LIN {X 0.103,Y -553.727,Z 590.333,A 0.000,B 0.000,C 90.000,E1 275.853} C_DIS
LIN {X 0.163,Y -552.917,Z 590.320,A 0.000,B 0.000,C 90.000,E1 273.612} C_DIS
LIN {X 0.102,Y -552.398,Z 590.309,A 0.000,B 0.000,C 90.000,E1 271.661} C_DIS
LIN {X -0.195,Y -552.147,Z 590.303,A 0.000,B 0.000,C 90.000,E1 270.573} C_DIS
LIN {X 0.184,Y -551.566,Z 590.294,A 0.000,B 0.000,C 90.000,E1 268.854} C_DIS
LIN {X 0.006,Y -550.867,Z 590.284,A 0.000,B 0.000,C 90.000,E1 267.192} C_DIS
LIN {X -0.206,Y -550.289,Z 590.277,A 0.000,B 0.000,C 90.000,E1 265.812} C_DIS
LIN {X 0.126,Y -549.551,Z 590.269,A 0.000,B 0.000,C 90.000,E1 264.375} C_DIS
LIN {X -0.148,Y -548.851,Z 590.263,A 0.000,B 0.000,C 90.000,E1 263.280} C_DIS
LIN {X 0.107,Y -547.994,Z 590.256,A 0.000,B 0.000,C 90.000,E1 262.129} C_DIS
LIN {X -0.025,Y -546.676,Z 590.249,A 0.000,B 0.000,C 90.000,E1 260.735} C_DIS
LIN {X 0.008,Y -544.774,Z 590.238,A 0.000,B 0.000,C 90.000,E1 258.757} C_DIS
LIN {X -0.079,Y -543.391,Z 590.230,A 0.000,B 0.000,C 90.000,E1 257.353} C_DIS
LIN {X 0.294,Y -541.048,Z 590.217,A 0.000,B 0.000,C 90.000,E1 255.046} C_DIS
LIN {X -0.049,Y -539.330,Z 590.208,A 0.000,B 0.000,C 90.000,E1 253.378} C_DIS
LIN {X 0.028,Y -537.748,Z 590.200,A 0.000,B 0.000,C 90.000,E1 251.945} C_DIS
LIN {X 0.200,Y -536.335,Z 590.193,A 0.000,B 0.000,C 90.000,E1 250.786} C_DIS
LIN {X 0.172,Y -534.674,Z 590.187,A 0.000,B 0.000,C 90.000,E1 249.645} C_DIS
LIN {X 0.288,Y -533.258,Z 590.182,A 0.000,B 0.000,C 90.000,E1 248.773} C_DIS
LIN {X 0.092,Y -530.601,Z 590.174,A 0.000,B 0.000,C 90.000,E1 247.358} C_DIS
LIN {X 0.227,Y -527.112,Z 590.165,A 0.000,B 0.000,C 90.000,E1 245.613} C_DIS
LIN {X 0.176,Y -524.691,Z 590.158,A 0.000,B 0.000,C 90.000,E1 244.460} C_DIS
LIN {X 0.245,Y -521.535,Z 590.150,A 0.000,B 0.000,C 90.000,E1 242.999} C_DIS
LIN {X 0.030,Y -518.163,Z 590.142,A 0.000,B 0.000,C 90.000,E1 241.563} C_DIS
LIN {X 0.098,Y -515.229,Z 590.136,A 0.000,B 0.000,C 90.000,E1 240.383} C_DIS
LIN {X 0.011,Y -509.881,Z 590.124,A 0.000,B 0.000,C 90.000,E1 238.329} C_DIS
LIN {X 0.105,Y -506.106,Z 590.116,A 0.000,B 0.000,C 90.000,E1 236.834} C_DIS
LIN {X -0.183,Y -502.744,Z 590.109,A 0.000,B 0.000,C 90.000,E1 235.674} C_DIS
LIN {X -0.116,Y -500.117,Z 590.104,A 0.000,B 0.000,C 90.000,E1 234.769} C_DIS
LIN {X 0.097,Y -492.736,Z 590.089,A 0.000,B 0.000,C 90.000,E1 232.029} C_DIS
LIN {X 0.027,Y -488.658,Z 590.081,A 0.000,B 0.000,C 90.000,E1 230.517} C_DIS
LIN {X -0.190,Y -484.697,Z 590.072,A 0.000,B 0.000,C 90.000,E1 229.013} C_DIS
LIN {X 0.093,Y -479.290,Z 590.060,A 0.000,B 0.000,C 90.000,E1 226.824} C_DIS
LIN {X -0.217,Y -474.782,Z 590.050,A 0.000,B 0.000,C 90.000,E1 225.000} C_DIS
LIN {X 0.185,Y -471.918,Z 590.043,A 0.000,B 0.000,C 90.000,E1 223.704} C_DIS
LIN {X 0.050,Y -467.520,Z 590.033,A 0.000,B 0.000,C 90.000,E1 221.838} C_DIS
LIN {X 0.112,Y -464.046,Z 590.024,A 0.000,B 0.000,C 90.000,E1 220.253} C_DIS
LIN {X 0.102,Y -460.700,Z 590.015,A 0.000,B 0.000,C 90.000,E1 218.669} C_DIS
LIN {X 0.094,Y -457.363,Z 590.006,A 0.000,B 0.000,C 90.000,E1 217.076} C_DIS
LIN {X -0.154,Y -453.442,Z 589.995,A 0.000,B 0.000,C 90.000,E1 215.185} C_DIS
LIN {X -0.110,Y -449.724,Z 589.985,A 0.000,B 0.000,C 90.000,E1 213.245} C_DIS
LIN {X -0.138,Y -443.891,Z 589.967,A 0.000,B 0.000,C 90.000,E1 210.001} C_DIS
LIN {X -0.203,Y -439.747,Z 589.954,A 0.000,B 0.000,C 90.000,E1 207.719} C_DIS
LIN {X -0.042,Y -436.870,Z 589.945,A 0.000,B 0.000,C 90.000,E1 206.052} C_DIS
LIN {X 0.098,Y -432.893,Z 589.932,A 0.000,B 0.000,C 90.000,E1 203.718} C_DIS
LIN {X 0.158,Y -428.613,Z 589.917,A 0.000,B 0.000,C 90.000,E1 201.046} C_DIS
LIN {X 0.166,Y -424.518,Z 589.902,A 0.000,B 0.000,C 90.000,E1 198.362} C_DIS
LIN {X 0.174,Y -420.785,Z 589.887,A 0.000,B 0.000,C 90.000,E1 195.662} C_DIS
LIN {X -0.186,Y -419.030,Z 589.880,A 0.000,B 0.000,C 90.000,E1 194.356} C_DIS
LIN {X 0.141,Y -417.098,Z 589.872,A 0.000,B 0.000,C 90.000,E1 192.952} C_DIS
LIN {X -0.146,Y -413.611,Z 589.859,A 0.000,B 0.000,C 90.000,E1 190.602} C_DIS
LIN {X 0.151,Y -410.179,Z 589.844,A 0.000,B 0.000,C 90.000,E1 187.814} C_DIS
LIN {X 0.197,Y -408.564,Z 589.836,A 0.000,B 0.000,C 90.000,E1 186.429} C_DIS
LIN {X 0.098,Y -404.784,Z 589.819,A 0.000,B 0.000,C 90.000,E1 183.326} C_DIS
LIN {X 0.160,Y -401.368,Z 589.797,A 0.000,B 0.000,C 90.000,E1 179.484} C_DIS
LIN {X -0.165,Y -399.570,Z 589.782,A 0.000,B 0.000,C 90.000,E1 176.731} C_DIS
LIN {X -0.089,Y -398.435,Z 589.766,A 0.000,B 0.000,C 90.000,E1 173.913} C_DIS
LIN {X 0.009,Y -397.785,Z 589.749,A 0.000,B 0.000,C 90.000,E1 170.735} C_DIS
LIN {X -0.126,Y -397.766,Z 589.731,A 0.000,B 0.000,C 90.000,E1 167.589} C_DIS
LIN {X 0.052,Y -398.187,Z 589.717,A 0.000,B 0.000,C 90.000,E1 165.102} C_DIS
LIN {X -0.064,Y -398.968,Z 589.702,A 0.000,B 0.000,C 90.000,E1 162.308} C_DIS
LIN {X 0.034,Y -399.714,Z 589.690,A 0.000,B 0.000,C 90.000,E1 160.188} C_DIS
LIN {X -0.168,Y -400.409,Z 589.680,A 0.000,B 0.000,C 90.000,E1 158.465} C_DIS
LIN {X -0.120,Y -401.392,Z 589.669,A 0.000,B 0.000,C 90.000,E1 156.357} C_DIS
LIN {X 0.102,Y -402.364,Z 589.657,A 0.000,B 0.000,C 90.000,E1 154.229} C_DIS
LIN {X -0.024,Y -403.383,Z 589.645,A 0.000,B 0.000,C 90.000,E1 152.153} C_DIS
LIN {X -0.024,Y -404.131,Z 589.636,A 0.000,B 0.000,C 90.000,E1 150.411} C_DIS
LIN {X 0.135,Y -404.680,Z 589.628,A 0.000,B 0.000,C 90.000,E1 148.997} C_DIS
LIN {X 0.213,Y -405.235,Z 589.618,A 0.000,B 0.000,C 90.000,E1 147.248} C_DIS
LIN {X 0.086,Y -405.715,Z 589.607,A 0.000,B 0.000,C 90.000,E1 145.182} C_DIS
LIN {X -0.031,Y -406.113,Z 589.597,A 0.000,B 0.000,C 90.000,E1 143.463} C_DIS
LIN {X 0.009,Y -406.580,Z 589.585,A 0.000,B 0.000,C 90.000,E1 141.376} C_DIS
LIN {X 0.156,Y -406.984,Z 589.576,A 0.000,B 0.000,C 90.000,E1 139.622} C_DIS
LIN {X 0.114,Y -407.316,Z 589.568,A 0.000,B 0.000,C 90.000,E1 138.243} C_DIS
LIN {X -0.240,Y -407.605,Z 589.557,A 0.000,B 0.000,C 90.000,E1 136.215} C_DIS
LIN {X 0.134,Y -407.816,Z 589.547,A 0.000,B 0.000,C 90.000,E1 134.433} C_DIS
LIN {X 0.071,Y -408.085,Z 589.535,A 0.000,B 0.000,C 90.000,E1 132.366} C_DIS
LIN {X 0.194,Y -408.172,Z 589.526,A 0.000,B 0.000,C 90.000,E1 130.620} C_DIS
LIN {X -0.092,Y -408.216,Z 589.518,A 0.000,B 0.000,C 90.000,E1 129.277} C_DIS
LIN {X 0.167,Y -408.231,Z 589.514,A 0.000,B 0.000,C 90.000,E1 128.463} C_DIS
LIN {X -0.072,Y -414.947,Z 589.501,A 0.000,B 0.000,C 90.000,E1 126.171} C_DIS
LIN {X 0.101,Y -415.909,Z 589.499,A 0.000,B 0.000,C 90.000,E1 125.804} C_DIS
LIN {X -0.016,Y -425.391,Z 589.478,A 0.000,B 0.000,C 90.000,E1 122.084} C_DIS
LIN {X -0.086,Y -428.983,Z 589.471,A 0.000,B 0.000,C 90.000,E1 120.875} C_DIS
LIN {X -0.125,Y -429.060,Z 589.471,A 0.000,B 0.000,C 90.000,E1 120.875} C_DIS
LIN {X 0.076,Y -438.663,Z 589.469,A 0.000,B 0.000,C 90.000,E1 120.413} C_DIS
LIN {X -0.052,Y -453.951,Z 589.465,A 0.000,B 0.000,C 90.000,E1 119.716} C_DIS
LIN {X 0.129,Y -467.535,Z 589.461,A 0.000,B 0.000,C 90.000,E1 119.027} C_DIS
LIN {X 0.032,Y -475.906,Z 589.459,A 0.000,B 0.000,C 90.000,E1 118.615} C_DIS
LIN {X -0.202,Y -485.846,Z 589.456,A 0.000,B 0.000,C 90.000,E1 118.103} C_DIS
LIN {X -0.052,Y -495.708,Z 589.453,A 0.000,B 0.000,C 90.000,E1 117.513} C_DIS
LIN {X -0.071,Y -502.085,Z 589.451,A 0.000,B 0.000,C 90.000,E1 117.129} C_DIS
LIN {X -0.060,Y -512.802,Z 589.447,A 0.000,B 0.000,C 90.000,E1 116.437} C_DIS
LIN {X 0.057,Y -517.558,Z 589.445,A 0.000,B 0.000,C 90.000,E1 116.104} C_DIS
LIN {X -0.067,Y -526.534,Z 589.441,A 0.000,B 0.000,C 90.000,E1 115.463} C_DIS
LIN {X 0.238,Y -533.686,Z 589.439,A 0.000,B 0.000,C 90.000,E1 114.899} C_DIS
LIN {X -0.150,Y -538.090,Z 589.437,A 0.000,B 0.000,C 90.000,E1 114.591} C_DIS
LIN {X 0.027,Y -544.873,Z 589.433,A 0.000,B 0.000,C 90.000,E1 114.003} C_DIS
LIN {X 0.244,Y -548.783,Z 589.432,A 0.000,B 0.000,C 90.000,E1 113.643} C_DIS
LIN {X -0.013,Y -554.752,Z 589.428,A 0.000,B 0.000,C 90.000,E1 113.078} C_DIS
LIN {X 0.050,Y -559.282,Z 589.426,A 0.000,B 0.000,C 90.000,E1 112.589} C_DIS
LIN {X 0.096,Y -564.684,Z 589.422,A 0.000,B 0.000,C 90.000,E1 111.897} C_DIS
LIN {X -0.075,Y -569.428,Z 589.418,A 0.000,B 0.000,C 90.000,E1 111.227} C_DIS
LIN {X -0.206,Y -573.566,Z 589.414,A 0.000,B 0.000,C 90.000,E1 110.556} C_DIS
LIN {X 0.078,Y -578.598,Z 589.409,A 0.000,B 0.000,C 90.000,E1 109.577} C_DIS
LIN {X -0.131,Y -583.212,Z 589.404,A 0.000,B 0.000,C 90.000,E1 108.652} C_DIS
LIN {X 0.147,Y -586.751,Z 589.399,A 0.000,B 0.000,C 90.000,E1 107.819} C_DIS
LIN {X 0.229,Y -588.912,Z 589.396,A 0.000,B 0.000,C 90.000,E1 107.275} C_DIS
LIN {X 0.009,Y -591.975,Z 589.392,A 0.000,B 0.000,C 90.000,E1 106.496} C_DIS
LIN {X 0.087,Y -595.800,Z 589.386,A 0.000,B 0.000,C 90.000,E1 105.426} C_DIS
LIN {X 0.220,Y -599.376,Z 589.380,A 0.000,B 0.000,C 90.000,E1 104.356} C_DIS
LIN {X 0.023,Y -605.560,Z 589.370,A 0.000,B 0.000,C 90.000,E1 102.535} C_DIS
LIN {X -0.031,Y -611.800,Z 589.360,A 0.000,B 0.000,C 90.000,E1 100.715} C_DIS
LIN {X -0.299,Y -614.429,Z 589.355,A 0.000,B 0.000,C 90.000,E1 99.962} C_DIS
LIN {X 0.196,Y -618.587,Z 589.348,A 0.000,B 0.000,C 90.000,E1 98.624} C_DIS
LIN {X 0.057,Y -622.599,Z 589.341,A 0.000,B 0.000,C 90.000,E1 97.352} C_DIS
LIN {X 0.211,Y -625.609,Z 589.335,A 0.000,B 0.000,C 90.000,E1 96.315} C_DIS
LIN {X 0.012,Y -627.702,Z 589.331,A 0.000,B 0.000,C 90.000,E1 95.568} C_DIS
LIN {X 0.236,Y -630.228,Z 589.325,A 0.000,B 0.000,C 90.000,E1 94.531} C_DIS
LIN {X -0.189,Y -632.360,Z 589.320,A 0.000,B 0.000,C 90.000,E1 93.555} C_DIS
LIN {X -0.214,Y -634.585,Z 589.313,A 0.000,B 0.000,C 90.000,E1 92.293} C_DIS
LIN {X 0.303,Y -635.778,Z 589.308,A 0.000,B 0.000,C 90.000,E1 91.489} C_DIS
LIN {X 0.049,Y -636.150,Z 589.307,A 0.000,B 0.000,C 90.000,E1 91.260} C_DIS
LIN {X 0.065,Y -637.392,Z 589.300,A 0.000,B 0.000,C 90.000,E1 90.000} C_DIS
LIN {X -0.041,Y -637.871,Z 589.296,A 0.000,B 0.000,C 90.000,E1 89.255} C_DIS
LIN {X -0.146,Y -638.129,Z 589.292,A 0.000,B 0.000,C 90.000,E1 88.511} C_DIS
LIN {X -0.229,Y -638.123,Z 589.288,A 0.000,B 0.000,C 90.000,E1 87.764} C_DIS
LIN {X 0.300,Y -637.875,Z 589.283,A 0.000,B 0.000,C 90.000,E1 86.963} C_DIS
LIN {X -0.034,Y -637.318,Z 589.278,A 0.000,B 0.000,C 90.000,E1 85.988} C_DIS
LIN {X 0.310,Y -636.408,Z 589.272,A 0.000,B 0.000,C 90.000,E1 84.951} C_DIS
LIN {X 0.017,Y -635.312,Z 589.267,A 0.000,B 0.000,C 90.000,E1 83.970} C_DIS
LIN {X -0.088,Y -634.277,Z 589.262,A 0.000,B 0.000,C 90.000,E1 83.223} C_DIS
LIN {X 0.217,Y -632.525,Z 589.257,A 0.000,B 0.000,C 90.000,E1 82.186} C_DIS
LIN {X -0.041,Y -630.463,Z 589.251,A 0.000,B 0.000,C 90.000,E1 81.197} C_DIS
LIN {X 0.302,Y -628.200,Z 589.245,A 0.000,B 0.000,C 90.000,E1 80.151} C_DIS
LIN {X -0.006,Y -625.708,Z 589.240,A 0.000,B 0.000,C 90.000,E1 79.162} C_DIS
LIN {X 0.046,Y -622.308,Z 589.233,A 0.000,B 0.000,C 90.000,E1 77.881} C_DIS
LIN {X 0.222,Y -620.910,Z 589.230,A 0.000,B 0.000,C 90.000,E1 77.353} C_DIS
LIN {X -0.286,Y -617.015,Z 589.223,A 0.000,B 0.000,C 90.000,E1 76.117} C_DIS
LIN {X -0.229,Y -614.491,Z 589.219,A 0.000,B 0.000,C 90.000,E1 75.338} C_DIS
LIN {X -0.005,Y -610.833,Z 589.213,A 0.000,B 0.000,C 90.000,E1 74.283} C_DIS
LIN {X -0.264,Y -606.705,Z 589.207,A 0.000,B 0.000,C 90.000,E1 73.268} C_DIS
LIN {X -0.304,Y -603.342,Z 589.203,A 0.000,B 0.000,C 90.000,E1 72.489} C_DIS
LIN {X -0.145,Y -600.317,Z 589.199,A 0.000,B 0.000,C 90.000,E1 71.819} C_DIS
LIN {X 0.202,Y -594.996,Z 589.193,A 0.000,B 0.000,C 90.000,E1 70.732} C_DIS
LIN {X 0.228,Y -590.658,Z 589.189,A 0.000,B 0.000,C 90.000,E1 69.934} C_DIS
LIN {X 0.013,Y -585.840,Z 589.184,A 0.000,B 0.000,C 90.000,E1 69.156} C_DIS
LIN {X 0.227,Y -581.416,Z 589.181,A 0.000,B 0.000,C 90.000,E1 68.465} C_DIS
LIN {X -0.271,Y -577.630,Z 589.178,A 0.000,B 0.000,C 90.000,E1 67.975} C_DIS
LIN {X -0.025,Y -572.375,Z 589.174,A 0.000,B 0.000,C 90.000,E1 67.283} C_DIS
LIN {X -0.251,Y -566.931,Z 589.170,A 0.000,B 0.000,C 90.000,E1 66.666} C_DIS
LIN {X 0.142,Y -563.380,Z 589.168,A 0.000,B 0.000,C 90.000,E1 66.230} C_DIS
LIN {X 0.231,Y -557.214,Z 589.165,A 0.000,B 0.000,C 90.000,E1 65.613} C_DIS
LIN {X -0.039,Y -552.060,Z 589.162,A 0.000,B 0.000,C 90.000,E1 65.177} C_DIS
LIN {X 0.031,Y -546.519,Z 589.160,A 0.000,B 0.000,C 90.000,E1 64.717} C_DIS
LIN {X -0.316,Y -541.738,Z 589.158,A 0.000,B 0.000,C 90.000,E1 64.409} C_DIS
LIN {X -0.139,Y -536.929,Z 589.156,A 0.000,B 0.000,C 90.000,E1 64.076} C_DIS
LIN {X 0.261,Y -530.053,Z 589.154,A 0.000,B 0.000,C 90.000,E1 63.640} C_DIS
LIN {X 0.086,Y -523.161,Z 589.152,A 0.000,B 0.000,C 90.000,E1 63.307} C_DIS
LIN {X -0.078,Y -516.360,Z 589.150,A 0.000,B 0.000,C 90.000,E1 62.999} C_DIS
LIN {X -0.092,Y -505.953,Z 589.147,A 0.000,B 0.000,C 90.000,E1 62.538} C_DIS
LIN {X -0.103,Y -492.338,Z 589.144,A 0.000,B 0.000,C 90.000,E1 61.948} C_DIS
LIN {X -0.006,Y -458.334,Z 589.136,A 0.000,B 0.000,C 90.000,E1 60.411} C_DIS
LIN {X -0.122,Y -450.998,Z 589.134,A 0.000,B 0.000,C 90.000,E1 60.049} C_DIS
LIN {X 0.226,Y -450.975,Z 589.134,A 0.000,B 0.000,C 90.000,E1 59.999} C_DIS
LIN {X 0.224,Y -444.233,Z 589.115,A 0.000,B 0.000,C 90.000,E1 56.628} C_DIS
LIN {X -0.087,Y -443.543,Z 589.113,A 0.000,B 0.000,C 90.000,E1 56.342} C_DIS
LIN {X -0.075,Y -434.458,Z 589.091,A 0.000,B 0.000,C 90.000,E1 52.396} C_DIS
LIN {X -0.070,Y -433.807,Z 589.089,A 0.000,B 0.000,C 90.000,E1 52.065} C_DIS
LIN {X -0.108,Y -433.823,Z 589.088,A 0.000,B 0.000,C 90.000,E1 51.904} C_DIS
LIN {X -0.028,Y -435.444,Z 589.078,A 0.000,B 0.000,C 90.000,E1 50.070} C_DIS
LIN {X 0.005,Y -437.214,Z 589.067,A 0.000,B 0.000,C 90.000,E1 48.081} C_DIS
LIN {X -0.011,Y -439.520,Z 589.052,A 0.000,B 0.000,C 90.000,E1 45.445} C_DIS
LIN {X 0.155,Y -440.657,Z 589.045,A 0.000,B 0.000,C 90.000,E1 44.109} C_DIS
LIN {X 0.022,Y -441.542,Z 589.038,A 0.000,B 0.000,C 90.000,E1 42.813} C_DIS
LIN {X -0.077,Y -442.261,Z 589.031,A 0.000,B 0.000,C 90.000,E1 41.515} C_DIS
LIN {X -0.130,Y -442.741,Z 589.025,A 0.000,B 0.000,C 90.000,E1 40.539} C_DIS
LIN {X -0.186,Y -443.365,Z 589.016,A 0.000,B 0.000,C 90.000,E1 38.910} C_DIS
LIN {X 0.119,Y -443.853,Z 589.007,A 0.000,B 0.000,C 90.000,E1 37.237} C_DIS
LIN {X -0.193,Y -444.089,Z 589.002,A 0.000,B 0.000,C 90.000,E1 36.297} C_DIS
LIN {X 0.214,Y -444.268,Z 588.992,A 0.000,B 0.000,C 90.000,E1 34.612} C_DIS
LIN {X 0.000,Y -444.218,Z 588.983,A 0.000,B 0.000,C 90.000,E1 33.007} C_DIS
LIN {X 0.027,Y -444.239,Z 588.971,A 0.000,B 0.000,C 90.000,E1 30.718} C_DIS
LIN {X 0.097,Y -444.213,Z 588.962,A 0.000,B 0.000,C 90.000,E1 29.077} C_DIS
LIN {X 0.012,Y -444.260,Z 588.951,A 0.000,B 0.000,C 90.000,E1 27.129} C_DIS
LIN {X -0.179,Y -444.308,Z 588.944,A 0.000,B 0.000,C 90.000,E1 25.848} C_DIS
LIN {X -0.112,Y -444.484,Z 588.934,A 0.000,B 0.000,C 90.000,E1 24.207} C_DIS
LIN {X -0.219,Y -444.728,Z 588.925,A 0.000,B 0.000,C 90.000,E1 22.589} C_DIS
LIN {X -0.047,Y -445.056,Z 588.914,A 0.000,B 0.000,C 90.000,E1 20.610} C_DIS
LIN {X 0.104,Y -445.449,Z 588.902,A 0.000,B 0.000,C 90.000,E1 18.308} C_DIS
LIN {X 0.132,Y -446.068,Z 588.889,A 0.000,B 0.000,C 90.000,E1 16.024} C_DIS
LIN {X -0.072,Y -446.918,Z 588.877,A 0.000,B 0.000,C 90.000,E1 13.772} C_DIS
LIN {X -0.180,Y -448.284,Z 588.862,A 0.000,B 0.000,C 90.000,E1 11.186} C_DIS
LIN {X 0.016,Y -449.845,Z 588.848,A 0.000,B 0.000,C 90.000,E1 8.568} C_DIS
LIN {X 0.122,Y -451.773,Z 588.833,A 0.000,B 0.000,C 90.000,E1 5.967} C_DIS
LIN {X 0.160,Y -454.081,Z 588.819,A 0.000,B 0.000,C 90.000,E1 3.383} C_DIS
LIN {X 0.070,Y -456.397,Z 588.806,A 0.000,B 0.000,C 90.000,E1 1.146} C_DIS
LIN {X -0.166,Y -459.209,Z 588.794,A 0.000,B 0.000,C 90.000,E1 358.854} C_DIS
LIN {X 0.091,Y -462.759,Z 588.779,A 0.000,B 0.000,C 90.000,E1 356.274} C_DIS
LIN {X -0.193,Y -466.009,Z 588.767,A 0.000,B 0.000,C 90.000,E1 354.090} C_DIS
LIN {X -0.104,Y -468.966,Z 588.757,A 0.000,B 0.000,C 90.000,E1 352.186} C_DIS
LIN {X 0.117,Y -471.829,Z 588.746,A 0.000,B 0.000,C 90.000,E1 350.274} C_DIS
LIN {X 0.019,Y -474.779,Z 588.736,A 0.000,B 0.000,C 90.000,E1 348.409} C_DIS
LIN {X 0.082,Y -477.877,Z 588.725,A 0.000,B 0.000,C 90.000,E1 346.533} C_DIS
LIN {X 0.011,Y -480.559,Z 588.717,A 0.000,B 0.000,C 90.000,E1 344.991} C_DIS
LIN {X -0.016,Y -484.658,Z 588.705,A 0.000,B 0.000,C 90.000,E1 342.834} C_DIS
LIN {X 0.082,Y -489.289,Z 588.691,A 0.000,B 0.000,C 90.000,E1 340.369} C_DIS
LIN {X 0.057,Y -492.236,Z 588.683,A 0.000,B 0.000,C 90.000,E1 338.847} C_DIS
LIN {X -0.148,Y -495.533,Z 588.672,A 0.000,B 0.000,C 90.000,E1 337.050} C_DIS
LIN {X -0.139,Y -498.127,Z 588.664,A 0.000,B 0.000,C 90.000,E1 335.537} C_DIS
LIN {X -0.141,Y -500.051,Z 588.657,A 0.000,B 0.000,C 90.000,E1 334.332} C_DIS
LIN {X -0.117,Y -501.996,Z 588.651,A 0.000,B 0.000,C 90.000,E1 333.127} C_DIS
LIN {X 0.025,Y -505.703,Z 588.637,A 0.000,B 0.000,C 90.000,E1 330.717} C_DIS
LIN {X -0.243,Y -508.962,Z 588.626,A 0.000,B 0.000,C 90.000,E1 328.663} C_DIS
LIN {X 0.196,Y -511.902,Z 588.616,A 0.000,B 0.000,C 90.000,E1 326.834} C_DIS
LIN {X 0.195,Y -515.529,Z 588.604,A 0.000,B 0.000,C 90.000,E1 324.769} C_DIS
LIN {X 0.154,Y -519.390,Z 588.593,A 0.000,B 0.000,C 90.000,E1 322.718} C_DIS
LIN {X -0.344,Y -523.881,Z 588.580,A 0.000,B 0.000,C 90.000,E1 320.436} C_DIS
LIN {X 0.128,Y -526.920,Z 588.572,A 0.000,B 0.000,C 90.000,E1 318.933} C_DIS
LIN {X -0.027,Y -529.247,Z 588.567,A 0.000,B 0.000,C 90.000,E1 318.081} C_DIS
LIN {X -0.322,Y -531.709,Z 588.563,A 0.000,B 0.000,C 90.000,E1 317.391} C_DIS
LIN {X -0.116,Y -534.196,Z 588.561,A 0.000,B 0.000,C 90.000,E1 316.905} C_DIS
LIN {X 0.070,Y -536.378,Z 588.559,A 0.000,B 0.000,C 90.000,E1 316.581} C_DIS
LIN {X 0.054,Y -538.214,Z 588.557,A 0.000,B 0.000,C 90.000,E1 316.296} C_DIS
LIN {X -0.273,Y -542.054,Z 588.555,A 0.000,B 0.000,C 90.000,E1 315.891} C_DIS
LIN {X 0.136,Y -546.676,Z 588.552,A 0.000,B 0.000,C 90.000,E1 315.405} C_DIS
LIN {X -0.087,Y -551.915,Z 588.550,A 0.000,B 0.000,C 90.000,E1 315.000} C_DIS
LIN {X 0.208,Y -566.862,Z 588.544,A 0.000,B 0.000,C 90.000,E1 313.866} C_DIS
LIN {X 0.158,Y -587.500,Z 588.536,A 0.000,B 0.000,C 90.000,E1 312.366} C_DIS
LIN {X -0.077,Y -593.270,Z 588.533,A 0.000,B 0.000,C 90.000,E1 311.962} C_DIS
LIN {X 0.100,Y -600.352,Z 588.530,A 0.000,B 0.000,C 90.000,E1 311.391} C_DIS
LIN {X -0.078,Y -604.427,Z 588.528,A 0.000,B 0.000,C 90.000,E1 311.067} C_DIS
LIN {X 0.064,Y -610.932,Z 588.525,A 0.000,B 0.000,C 90.000,E1 310.458} C_DIS
LIN {X 0.040,Y -613.520,Z 588.523,A 0.000,B 0.000,C 90.000,E1 310.216} C_DIS
LIN {X -0.290,Y -619.311,Z 588.520,A 0.000,B 0.000,C 90.000,E1 309.644} C_DIS
LIN {X 0.137,Y -623.800,Z 588.517,A 0.000,B 0.000,C 90.000,E1 309.116} C_DIS
LIN {X -0.138,Y -630.493,Z 588.513,A 0.000,B 0.000,C 90.000,E1 308.382} C_DIS
LIN {X -0.048,Y -638.673,Z 588.508,A 0.000,B 0.000,C 90.000,E1 307.363} C_DIS
LIN {X -0.155,Y -642.541,Z 588.505,A 0.000,B 0.000,C 90.000,E1 306.870} C_DIS
LIN {X -0.235,Y -646.121,Z 588.502,A 0.000,B 0.000,C 90.000,E1 306.377} C_DIS
LIN {X -0.190,Y -651.020,Z 588.498,A 0.000,B 0.000,C 90.000,E1 305.644} C_DIS
LIN {X 0.318,Y -654.104,Z 588.495,A 0.000,B 0.000,C 90.000,E1 305.105} C_DIS
LIN {X 0.275,Y -656.265,Z 588.493,A 0.000,B 0.000,C 90.000,E1 304.739} C_DIS
LIN {X 0.332,Y -659.571,Z 588.490,A 0.000,B 0.000,C 90.000,E1 304.119} C_DIS
LIN {X -0.003,Y -662.000,Z 588.487,A 0.000,B 0.000,C 90.000,E1 303.658} C_DIS
LIN {X -0.393,Y -665.301,Z 588.483,A 0.000,B 0.000,C 90.000,E1 302.959} C_DIS
LIN {X -0.197,Y -668.414,Z 588.479,A 0.000,B 0.000,C 90.000,E1 302.212} C_DIS
LIN {X 0.189,Y -672.332,Z 588.474,A 0.000,B 0.000,C 90.000,E1 301.209} C_DIS
LIN {X 0.047,Y -676.130,Z 588.468,A 0.000,B 0.000,C 90.000,E1 300.256} C_DIS
LIN {X 0.197,Y -679.703,Z 588.463,A 0.000,B 0.000,C 90.000,E1 299.283} C_DIS
LIN {X -0.199,Y -683.002,Z 588.458,A 0.000,B 0.000,C 90.000,E1 298.359} C_DIS
LIN {X 0.262,Y -686.713,Z 588.451,A 0.000,B 0.000,C 90.000,E1 297.129} C_DIS
LIN {X 0.014,Y -688.584,Z 588.447,A 0.000,B 0.000,C 90.000,E1 296.437} C_DIS
LIN {X -0.373,Y -688.952,Z 588.446,A 0.000,B 0.000,C 90.000,E1 296.232} C_DIS
LIN {X 0.089,Y -689.180,Z 588.443,A 0.000,B 0.000,C 90.000,E1 295.720} C_DIS
LIN {X 0.321,Y -688.932,Z 588.442,A 0.000,B 0.000,C 90.000,E1 295.463} C_DIS
LIN {X -0.132,Y -687.243,Z 588.439,A 0.000,B 0.000,C 90.000,E1 295.027} C_DIS
LIN {X -0.018,Y -686.727,Z 588.438,A 0.000,B 0.000,C 90.000,E1 294.899} C_DIS
LIN {X 0.096,Y -685.999,Z 588.438,A 0.000,B 0.000,C 90.000,E1 294.771} C_DIS
LIN {X 0.206,Y -684.865,Z 588.437,A 0.000,B 0.000,C 90.000,E1 294.643} C_DIS
LIN {X 0.313,Y -680.019,Z 588.435,A 0.000,B 0.000,C 90.000,E1 294.207} C_DIS
LIN {X -0.121,Y -678.129,Z 588.434,A 0.000,B 0.000,C 90.000,E1 294.131} C_DIS
LIN {X -0.045,Y -670.038,Z 588.432,A 0.000,B 0.000,C 90.000,E1 293.823} C_DIS
LIN {X -0.184,Y -667.501,Z 588.432,A 0.000,B 0.000,C 90.000,E1 293.770} C_DIS
LIN {X -0.305,Y -661.294,Z 588.431,A 0.000,B 0.000,C 90.000,E1 293.643} C_DIS
LIN {X 0.269,Y -638.978,Z 588.429,A 0.000,B 0.000,C 90.000,E1 293.206} C_DIS
LIN {X -0.018,Y -629.598,Z 588.428,A 0.000,B 0.000,C 90.000,E1 293.025} C_DIS
LIN {X -0.193,Y -616.215,Z 588.426,A 0.000,B 0.000,C 90.000,E1 292.695} C_DIS
LIN {X -0.203,Y -595.903,Z 588.423,A 0.000,B 0.000,C 90.000,E1 292.078} C_DIS
LIN {X 0.143,Y -578.394,Z 588.419,A 0.000,B 0.000,C 90.000,E1 291.482} C_DIS
LIN {X 0.025,Y -571.534,Z 588.418,A 0.000,B 0.000,C 90.000,E1 291.280} C_DIS
LIN {X -0.186,Y -566.448,Z 588.417,A 0.000,B 0.000,C 90.000,E1 291.099} C_DIS
LIN {X 0.220,Y -561.824,Z 588.416,A 0.000,B 0.000,C 90.000,E1 290.791} C_DIS
LIN {X 0.191,Y -561.777,Z 588.416,A 0.000,B 0.000,C 90.000,E1 290.791} C_DIS
LIN {X 0.127,Y -560.661,Z 588.415,A 0.000,B 0.000,C 90.000,E1 290.610} C_DIS
LIN {X 0.085,Y -560.646,Z 588.415,A 0.000,B 0.000,C 90.000,E1 290.610} C_DIS
LIN {X 0.204,Y -560.137,Z 588.412,A 0.000,B 0.000,C 90.000,E1 290.174} C_DIS
LIN {X -0.104,Y -560.141,Z 588.405,A 0.000,B 0.000,C 90.000,E1 288.833} C_DIS
LIN {X 0.222,Y -559.944,Z 588.398,A 0.000,B 0.000,C 90.000,E1 287.692} C_DIS
LIN {X -0.258,Y -559.330,Z 588.389,A 0.000,B 0.000,C 90.000,E1 286.079} C_DIS
LIN {X -0.094,Y -558.821,Z 588.383,A 0.000,B 0.000,C 90.000,E1 284.954} C_DIS
LIN {X 0.203,Y -558.108,Z 588.375,A 0.000,B 0.000,C 90.000,E1 283.536} C_DIS
LIN {X 0.210,Y -556.977,Z 588.365,A 0.000,B 0.000,C 90.000,E1 281.591} C_DIS
LIN {X -0.043,Y -555.897,Z 588.354,A 0.000,B 0.000,C 90.000,E1 279.670} C_DIS
LIN {X 0.140,Y -554.864,Z 588.343,A 0.000,B 0.000,C 90.000,E1 277.701} C_DIS
LIN {X 0.227,Y -553.938,Z 588.332,A 0.000,B 0.000,C 90.000,E1 275.739} C_DIS
LIN {X -0.192,Y -553.091,Z 588.318,A 0.000,B 0.000,C 90.000,E1 273.269} C_DIS
LIN {X -0.245,Y -552.583,Z 588.307,A 0.000,B 0.000,C 90.000,E1 271.318} C_DIS
LIN {X 0.079,Y -552.175,Z 588.299,A 0.000,B 0.000,C 90.000,E1 269.885} C_DIS
LIN {X -0.157,Y -551.621,Z 588.292,A 0.000,B 0.000,C 90.000,E1 268.511} C_DIS
LIN {X 0.101,Y -551.168,Z 588.285,A 0.000,B 0.000,C 90.000,E1 267.364} C_DIS
LIN {X -0.052,Y -550.490,Z 588.276,A 0.000,B 0.000,C 90.000,E1 265.698} C_DIS
LIN {X -0.267,Y -549.745,Z 588.268,A 0.000,B 0.000,C 90.000,E1 264.318} C_DIS
LIN {X 0.007,Y -549.039,Z 588.262,A 0.000,B 0.000,C 90.000,E1 263.166} C_DIS
LIN {X -0.206,Y -548.177,Z 588.256,A 0.000,B 0.000,C 90.000,E1 262.064} C_DIS
LIN {X 0.129,Y -546.783,Z 588.248,A 0.000,B 0.000,C 90.000,E1 260.622} C_DIS
LIN {X 0.169,Y -545.194,Z 588.239,A 0.000,B 0.000,C 90.000,E1 258.926} C_DIS
LIN {X 0.097,Y -543.810,Z 588.231,A 0.000,B 0.000,C 90.000,E1 257.521} C_DIS
LIN {X -0.088,Y -542.575,Z 588.224,A 0.000,B 0.000,C 90.000,E1 256.408} C_DIS
LIN {X -0.020,Y -540.884,Z 588.215,A 0.000,B 0.000,C 90.000,E1 254.700} C_DIS
LIN {X 0.298,Y -539.103,Z 588.206,A 0.000,B 0.000,C 90.000,E1 252.960} C_DIS
LIN {X -0.190,Y -537.830,Z 588.199,A 0.000,B 0.000,C 90.000,E1 251.873} C_DIS
LIN {X -0.187,Y -536.375,Z 588.193,A 0.000,B 0.000,C 90.000,E1 250.732} C_DIS
LIN {X -0.031,Y -534.658,Z 588.187,A 0.000,B 0.000,C 90.000,E1 249.571} C_DIS
LIN {X -0.103,Y -533.184,Z 588.182,A 0.000,B 0.000,C 90.000,E1 248.720} C_DIS
LIN {X 0.001,Y -531.609,Z 588.177,A 0.000,B 0.000,C 90.000,E1 247.847} C_DIS
LIN {X 0.282,Y -529.345,Z 588.171,A 0.000,B 0.000,C 90.000,E1 246.666} C_DIS
LIN {X -0.088,Y -525.828,Z 588.161,A 0.000,B 0.000,C 90.000,E1 244.973} C_DIS
LIN {X 0.153,Y -522.046,Z 588.151,A 0.000,B 0.000,C 90.000,E1 243.204} C_DIS
LIN {X -0.058,Y -518.655,Z 588.143,A 0.000,B 0.000,C 90.000,E1 241.769} C_DIS
LIN {X 0.100,Y -516.477,Z 588.138,A 0.000,B 0.000,C 90.000,E1 240.873} C_DIS
LIN {X -0.053,Y -513.450,Z 588.132,A 0.000,B 0.000,C 90.000,E1 239.715} C_DIS
LIN {X -0.185,Y -508.111,Z 588.120,A 0.000,B 0.000,C 90.000,E1 237.661} C_DIS
LIN {X -0.060,Y -505.781,Z 588.115,A 0.000,B 0.000,C 90.000,E1 236.755} C_DIS
LIN {X -0.238,Y -503.290,Z 588.110,A 0.000,B 0.000,C 90.000,E1 235.881} C_DIS
LIN {X -0.165,Y -500.688,Z 588.105,A 0.000,B 0.000,C 90.000,E1 234.975} C_DIS
LIN {X -0.073,Y -492.444,Z 588.089,A 0.000,B 0.000,C 90.000,E1 231.949} C_DIS
LIN {X -0.016,Y -486.005,Z 588.075,A 0.000,B 0.000,C 90.000,E1 229.504} C_DIS
LIN {X -0.212,Y -479.765,Z 588.061,A 0.000,B 0.000,C 90.000,E1 227.067} C_DIS
LIN {X -0.067,Y -474.482,Z 588.049,A 0.000,B 0.000,C 90.000,E1 224.879} C_DIS
LIN {X -0.004,Y -471.586,Z 588.042,A 0.000,B 0.000,C 90.000,E1 223.623} C_DIS
LIN {X -0.075,Y -466.498,Z 588.030,A 0.000,B 0.000,C 90.000,E1 221.434} C_DIS
LIN {X 0.113,Y -461.741,Z 588.018,A 0.000,B 0.000,C 90.000,E1 219.197} C_DIS
LIN {X -0.131,Y -457.761,Z 588.007,A 0.000,B 0.000,C 90.000,E1 217.317} C_DIS
LIN {X 0.256,Y -453.149,Z 587.995,A 0.000,B 0.000,C 90.000,E1 215.025} C_DIS
LIN {X -0.016,Y -448.790,Z 587.982,A 0.000,B 0.000,C 90.000,E1 212.801} C_DIS
LIN {X -0.062,Y -444.133,Z 587.968,A 0.000,B 0.000,C 90.000,E1 210.207} C_DIS
LIN {X 0.047,Y -440.587,Z 587.957,A 0.000,B 0.000,C 90.000,E1 208.231} C_DIS
LIN {X -0.171,Y -437.710,Z 587.948,A 0.000,B 0.000,C 90.000,E1 206.616} C_DIS
LIN {X 0.163,Y -434.263,Z 587.937,A 0.000,B 0.000,C 90.000,E1 204.591} C_DIS
LIN {X 0.201,Y -432.053,Z 587.929,A 0.000,B 0.000,C 90.000,E1 203.259} C_DIS
LIN {X -0.146,Y -428.318,Z 587.916,A 0.000,B 0.000,C 90.000,E1 200.972} C_DIS
LIN {X 0.056,Y -424.773,Z 587.903,A 0.000,B 0.000,C 90.000,E1 198.598} C_DIS
LIN {X 0.128,Y -420.596,Z 587.887,A 0.000,B 0.000,C 90.000,E1 195.552} C_DIS
LIN {X -0.230,Y -418.833,Z 587.879,A 0.000,B 0.000,C 90.000,E1 194.245} C_DIS
LIN {X 0.192,Y -416.889,Z 587.871,A 0.000,B 0.000,C 90.000,E1 192.827} C_DIS
LIN {X 0.175,Y -413.909,Z 587.860,A 0.000,B 0.000,C 90.000,E1 190.782} C_DIS
LIN {X 0.113,Y -410.041,Z 587.843,A 0.000,B 0.000,C 90.000,E1 187.701} C_DIS
LIN {X 0.160,Y -408.422,Z 587.835,A 0.000,B 0.000,C 90.000,E1 186.315} C_DIS
LIN {X 0.118,Y -405.879,Z 587.824,A 0.000,B 0.000,C 90.000,E1 184.245} C_DIS
LIN {X 0.161,Y -401.618,Z 587.799,A 0.000,B 0.000,C 90.000,E1 179.714} C_DIS
LIN {X -0.177,Y -399.806,Z 587.783,A 0.000,B 0.000,C 90.000,E1 176.963} C_DIS
LIN {X -0.130,Y -398.491,Z 587.766,A 0.000,B 0.000,C 90.000,E1 173.799} C_DIS
LIN {X -0.012,Y -397.940,Z 587.750,A 0.000,B 0.000,C 90.000,E1 170.971} C_DIS
LIN {X -0.122,Y -397.811,Z 587.734,A 0.000,B 0.000,C 90.000,E1 168.173} C_DIS
LIN {X -0.039,Y -398.192,Z 587.721,A 0.000,B 0.000,C 90.000,E1 165.700} C_DIS
LIN {X -0.118,Y -398.775,Z 587.707,A 0.000,B 0.000,C 90.000,E1 163.251} C_DIS
LIN {X -0.139,Y -399.499,Z 587.695,A 0.000,B 0.000,C 90.000,E1 161.148} C_DIS
LIN {X -0.025,Y -400.331,Z 587.684,A 0.000,B 0.000,C 90.000,E1 159.028} C_DIS
LIN {X 0.094,Y -401.465,Z 587.670,A 0.000,B 0.000,C 90.000,E1 156.561} C_DIS
LIN {X 0.121,Y -402.463,Z 587.658,A 0.000,B 0.000,C 90.000,E1 154.460} C_DIS
LIN {X 0.180,Y -403.475,Z 587.647,A 0.000,B 0.000,C 90.000,E1 152.359} C_DIS
LIN {X -0.172,Y -404.269,Z 587.637,A 0.000,B 0.000,C 90.000,E1 150.667} C_DIS
LIN {X -0.105,Y -404.972,Z 587.627,A 0.000,B 0.000,C 90.000,E1 148.918} C_DIS
LIN {X -0.112,Y -405.597,Z 587.616,A 0.000,B 0.000,C 90.000,E1 146.834} C_DIS
LIN {X 0.001,Y -406.072,Z 587.604,A 0.000,B 0.000,C 90.000,E1 144.736} C_DIS
LIN {X -0.020,Y -406.440,Z 587.594,A 0.000,B 0.000,C 90.000,E1 143.004} C_DIS
LIN {X 0.096,Y -406.994,Z 587.581,A 0.000,B 0.000,C 90.000,E1 140.561} C_DIS
LIN {X 0.081,Y -407.443,Z 587.569,A 0.000,B 0.000,C 90.000,E1 138.485} C_DIS
LIN {X 0.008,Y -407.721,Z 587.558,A 0.000,B 0.000,C 90.000,E1 136.419} C_DIS
LIN {X 0.102,Y -407.938,Z 587.548,A 0.000,B 0.000,C 90.000,E1 134.676} C_DIS
LIN {X -0.112,Y -408.249,Z 587.535,A 0.000,B 0.000,C 90.000,E1 132.285} C_DIS
LIN {X 0.163,Y -408.354,Z 587.523,A 0.000,B 0.000,C 90.000,E1 130.172} C_DIS
LIN {X 0.030,Y -408.284,Z 587.514,A 0.000,B 0.000,C 90.000,E1 128.463} C_DIS
LIN {X 0.013,Y -415.406,Z 587.500,A 0.000,B 0.000,C 90.000,E1 126.011} C_DIS
LIN {X 0.074,Y -425.807,Z 587.477,A 0.000,B 0.000,C 90.000,E1 121.926} C_DIS
LIN {X 0.022,Y -429.816,Z 587.470,A 0.000,B 0.000,C 90.000,E1 120.590} C_DIS
LIN {X -0.014,Y -429.872,Z 587.470,A 0.000,B 0.000,C 90.000,E1 120.590} C_DIS
LIN {X 0.019,Y -437.258,Z 587.468,A 0.000,B 0.000,C 90.000,E1 120.256} C_DIS
LIN {X 0.023,Y -454.334,Z 587.464,A 0.000,B 0.000,C 90.000,E1 119.461} C_DIS
LIN {X -0.163,Y -467.918,Z 587.460,A 0.000,B 0.000,C 90.000,E1 118.821} C_DIS
LIN {X 0.070,Y -478.033,Z 587.457,A 0.000,B 0.000,C 90.000,E1 118.281} C_DIS
LIN {X -0.169,Y -484.347,Z 587.455,A 0.000,B 0.000,C 90.000,E1 117.975} C_DIS
LIN {X 0.084,Y -494.131,Z 587.452,A 0.000,B 0.000,C 90.000,E1 117.385} C_DIS
LIN {X 0.191,Y -500.490,Z 587.450,A 0.000,B 0.000,C 90.000,E1 117.001} C_DIS
LIN {X 0.137,Y -509.934,Z 587.447,A 0.000,B 0.000,C 90.000,E1 116.411} C_DIS
LIN {X -0.051,Y -517.628,Z 587.444,A 0.000,B 0.000,C 90.000,E1 115.924} C_DIS
LIN {X 0.197,Y -528.051,Z 587.440,A 0.000,B 0.000,C 90.000,E1 115.155} C_DIS
LIN {X 0.176,Y -533.889,Z 587.438,A 0.000,B 0.000,C 90.000,E1 114.719} C_DIS
LIN {X 0.024,Y -538.414,Z 587.436,A 0.000,B 0.000,C 90.000,E1 114.387} C_DIS
LIN {X -0.088,Y -545.311,Z 587.432,A 0.000,B 0.000,C 90.000,E1 113.823} C_DIS
LIN {X 0.034,Y -548.183,Z 587.431,A 0.000,B 0.000,C 90.000,E1 113.567} C_DIS
LIN {X -0.064,Y -553.441,Z 587.428,A 0.000,B 0.000,C 90.000,E1 113.078} C_DIS
LIN {X 0.326,Y -558.519,Z 587.425,A 0.000,B 0.000,C 90.000,E1 112.514} C_DIS
LIN {X -0.262,Y -564.071,Z 587.422,A 0.000,B 0.000,C 90.000,E1 111.897} C_DIS
LIN {X 0.088,Y -568.975,Z 587.418,A 0.000,B 0.000,C 90.000,E1 111.173} C_DIS
LIN {X 0.159,Y -573.241,Z 587.414,A 0.000,B 0.000,C 90.000,E1 110.482} C_DIS
LIN {X -0.024,Y -577.702,Z 587.409,A 0.000,B 0.000,C 90.000,E1 109.685} C_DIS
LIN {X -0.277,Y -581.169,Z 587.406,A 0.000,B 0.000,C 90.000,E1 109.033} C_DIS
LIN {X -0.307,Y -584.388,Z 587.402,A 0.000,B 0.000,C 90.000,E1 108.362} C_DIS
LIN {X -0.083,Y -588.470,Z 587.397,A 0.000,B 0.000,C 90.000,E1 107.402} C_DIS
LIN {X 0.117,Y -592.642,Z 587.391,A 0.000,B 0.000,C 90.000,E1 106.315} C_DIS
LIN {X -0.229,Y -595.634,Z 587.386,A 0.000,B 0.000,C 90.000,E1 105.552} C_DIS
LIN {X -0.095,Y -599.285,Z 587.380,A 0.000,B 0.000,C 90.000,E1 104.481} C_DIS
LIN {X -0.154,Y -605.572,Z 587.370,A 0.000,B 0.000,C 90.000,E1 102.647} C_DIS
LIN {X -0.076,Y -610.968,Z 587.362,A 0.000,B 0.000,C 90.000,E1 101.074} C_DIS
LIN {X -0.236,Y -615.401,Z 587.354,A 0.000,B 0.000,C 90.000,E1 99.792} C_DIS
LIN {X -0.090,Y -618.794,Z 587.349,A 0.000,B 0.000,C 90.000,E1 98.746} C_DIS
LIN {X -0.138,Y -622.873,Z 587.341,A 0.000,B 0.000,C 90.000,E1 97.466} C_DIS
LIN {X 0.248,Y -625.198,Z 587.337,A 0.000,B 0.000,C 90.000,E1 96.663} C_DIS
LIN {X -0.181,Y -628.082,Z 587.332,A 0.000,B 0.000,C 90.000,E1 95.682} C_DIS
LIN {X 0.273,Y -630.067,Z 587.327,A 0.000,B 0.000,C 90.000,E1 94.878} C_DIS
LIN {X 0.123,Y -631.825,Z 587.323,A 0.000,B 0.000,C 90.000,E1 94.131} C_DIS
LIN {X -0.241,Y -633.809,Z 587.317,A 0.000,B 0.000,C 90.000,E1 93.151} C_DIS
LIN {X -0.016,Y -635.587,Z 587.312,A 0.000,B 0.000,C 90.000,E1 92.121} C_DIS
LIN {X -0.124,Y -636.742,Z 587.308,A 0.000,B 0.000,C 90.000,E1 91.375} C_DIS
LIN {X -0.099,Y -638.073,Z 587.301,A 0.000,B 0.000,C 90.000,E1 90.115} C_DIS
LIN {X -0.199,Y -638.572,Z 587.296,A 0.000,B 0.000,C 90.000,E1 89.370} C_DIS
LIN {X -0.296,Y -638.850,Z 587.292,A 0.000,B 0.000,C 90.000,E1 88.625} C_DIS
LIN {X 0.267,Y -638.875,Z 587.288,A 0.000,B 0.000,C 90.000,E1 87.822} C_DIS
LIN {X 0.166,Y -638.646,Z 587.284,A 0.000,B 0.000,C 90.000,E1 87.078} C_DIS
LIN {X -0.156,Y -638.092,Z 587.278,A 0.000,B 0.000,C 90.000,E1 86.102} C_DIS
LIN {X -0.233,Y -637.443,Z 587.274,A 0.000,B 0.000,C 90.000,E1 85.355} C_DIS
LIN {X -0.147,Y -636.065,Z 587.267,A 0.000,B 0.000,C 90.000,E1 84.090} C_DIS
LIN {X -0.176,Y -635.087,Z 587.263,A 0.000,B 0.000,C 90.000,E1 83.337} C_DIS
LIN {X 0.143,Y -633.288,Z 587.257,A 0.000,B 0.000,C 90.000,E1 82.299} C_DIS
LIN {X 0.093,Y -631.815,Z 587.253,A 0.000,B 0.000,C 90.000,E1 81.546} C_DIS
LIN {X 0.149,Y -628.972,Z 587.246,A 0.000,B 0.000,C 90.000,E1 80.274} C_DIS
LIN {X 0.164,Y -627.082,Z 587.242,A 0.000,B 0.000,C 90.000,E1 79.511} C_DIS
LIN {X -0.159,Y -624.413,Z 587.236,A 0.000,B 0.000,C 90.000,E1 78.522} C_DIS
LIN {X 0.000,Y -620.807,Z 587.229,A 0.000,B 0.000,C 90.000,E1 77.229} C_DIS
LIN {X 0.097,Y -616.802,Z 587.222,A 0.000,B 0.000,C 90.000,E1 75.936} C_DIS
LIN {X -0.002,Y -614.155,Z 587.218,A 0.000,B 0.000,C 90.000,E1 75.172} C_DIS
LIN {X 0.030,Y -611.332,Z 587.213,A 0.000,B 0.000,C 90.000,E1 74.393} C_DIS
LIN {X 0.120,Y -609.273,Z 587.210,A 0.000,B 0.000,C 90.000,E1 73.866} C_DIS
LIN {X -0.217,Y -607.170,Z 587.208,A 0.000,B 0.000,C 90.000,E1 73.378} C_DIS
LIN {X 0.283,Y -603.117,Z 587.203,A 0.000,B 0.000,C 90.000,E1 72.417} C_DIS
LIN {X 0.253,Y -600.034,Z 587.199,A 0.000,B 0.000,C 90.000,E1 71.764} C_DIS
LIN {X 0.149,Y -594.615,Z 587.193,A 0.000,B 0.000,C 90.000,E1 70.732} C_DIS
LIN {X 0.241,Y -590.173,Z 587.189,A 0.000,B 0.000,C 90.000,E1 69.934} C_DIS
LIN {X -0.102,Y -586.202,Z 587.185,A 0.000,B 0.000,C 90.000,E1 69.316} C_DIS
LIN {X -0.089,Y -581.704,Z 587.181,A 0.000,B 0.000,C 90.000,E1 68.646} C_DIS
LIN {X -0.122,Y -576.771,Z 587.178,A 0.000,B 0.000,C 90.000,E1 67.975} C_DIS
LIN {X -0.333,Y -572.726,Z 587.175,A 0.000,B 0.000,C 90.000,E1 67.486} C_DIS
LIN {X -0.138,Y -568.090,Z 587.172,A 0.000,B 0.000,C 90.000,E1 66.922} C_DIS
LIN {X 0.043,Y -563.109,Z 587.169,A 0.000,B 0.000,C 90.000,E1 66.357} C_DIS
LIN {X -0.107,Y -557.740,Z 587.166,A 0.000,B 0.000,C 90.000,E1 65.845} C_DIS
LIN {X -0.186,Y -552.057,Z 587.163,A 0.000,B 0.000,C 90.000,E1 65.357} C_DIS
LIN {X 0.273,Y -546.223,Z 587.160,A 0.000,B 0.000,C 90.000,E1 64.845} C_DIS
LIN {X 0.101,Y -541.578,Z 587.159,A 0.000,B 0.000,C 90.000,E1 64.537} C_DIS
LIN {X 0.034,Y -536.627,Z 587.157,A 0.000,B 0.000,C 90.000,E1 64.229} C_DIS
LIN {X 0.060,Y -529.887,Z 587.155,A 0.000,B 0.000,C 90.000,E1 63.845} C_DIS
LIN {X -0.064,Y -523.021,Z 587.153,A 0.000,B 0.000,C 90.000,E1 63.512} C_DIS
LIN {X -0.266,Y -514.316,Z 587.151,A 0.000,B 0.000,C 90.000,E1 63.127} C_DIS
LIN {X -0.210,Y -505.688,Z 587.148,A 0.000,B 0.000,C 90.000,E1 62.743} C_DIS
LIN {X -0.159,Y -491.974,Z 587.145,A 0.000,B 0.000,C 90.000,E1 62.153} C_DIS
LIN {X -0.119,Y -459.751,Z 587.137,A 0.000,B 0.000,C 90.000,E1 60.717} C_DIS
LIN {X 0.081,Y -451.667,Z 587.135,A 0.000,B 0.000,C 90.000,E1 60.284} C_DIS
LIN {X 0.038,Y -451.572,Z 587.135,A 0.000,B 0.000,C 90.000,E1 60.284} C_DIS
LIN {X 0.049,Y -444.194,Z 587.115,A 0.000,B 0.000,C 90.000,E1 56.628} C_DIS
LIN {X 0.108,Y -443.483,Z 587.113,A 0.000,B 0.000,C 90.000,E1 56.294} C_DIS
LIN {X -0.236,Y -434.167,Z 587.090,A 0.000,B 0.000,C 90.000,E1 52.271} C_DIS
LIN {X 0.059,Y -434.112,Z 587.090,A 0.000,B 0.000,C 90.000,E1 52.190} C_DIS
LIN {X -0.191,Y -436.088,Z 587.078,A 0.000,B 0.000,C 90.000,E1 50.070} C_DIS
LIN {X -0.143,Y -437.916,Z 587.067,A 0.000,B 0.000,C 90.000,E1 48.081} C_DIS
LIN {X 0.206,Y -439.989,Z 587.054,A 0.000,B 0.000,C 90.000,E1 45.729} C_DIS
LIN {X 0.071,Y -441.162,Z 587.047,A 0.000,B 0.000,C 90.000,E1 44.433} C_DIS
LIN {X -0.051,Y -442.130,Z 587.040,A 0.000,B 0.000,C 90.000,E1 43.137} C_DIS
LIN {X -0.139,Y -442.893,Z 587.032,A 0.000,B 0.000,C 90.000,E1 41.838} C_DIS
LIN {X -0.213,Y -443.520,Z 587.025,A 0.000,B 0.000,C 90.000,E1 40.539} C_DIS
LIN {X 0.060,Y -444.042,Z 587.018,A 0.000,B 0.000,C 90.000,E1 39.197} C_DIS
LIN {X 0.064,Y -444.456,Z 587.011,A 0.000,B 0.000,C 90.000,E1 37.890} C_DIS
LIN {X 0.074,Y -444.782,Z 587.003,A 0.000,B 0.000,C 90.000,E1 36.583} C_DIS
LIN {X 0.131,Y -444.921,Z 586.994,A 0.000,B 0.000,C 90.000,E1 34.945} C_DIS
LIN {X -0.007,Y -444.905,Z 586.987,A 0.000,B 0.000,C 90.000,E1 33.658} C_DIS
LIN {X 0.227,Y -444.815,Z 586.976,A 0.000,B 0.000,C 90.000,E1 31.671} C_DIS
LIN {X -0.074,Y -444.820,Z 586.967,A 0.000,B 0.000,C 90.000,E1 30.079} C_DIS
LIN {X 0.075,Y -444.772,Z 586.956,A 0.000,B 0.000,C 90.000,E1 28.103} C_DIS
LIN {X 0.000,Y -444.817,Z 586.945,A 0.000,B 0.000,C 90.000,E1 26.155} C_DIS
LIN {X -0.068,Y -444.938,Z 586.935,A 0.000,B 0.000,C 90.000,E1 24.207} C_DIS
LIN {X -0.166,Y -445.155,Z 586.925,A 0.000,B 0.000,C 90.000,E1 22.589} C_DIS
LIN {X 0.016,Y -445.439,Z 586.915,A 0.000,B 0.000,C 90.000,E1 20.610} C_DIS
LIN {X -0.245,Y -445.805,Z 586.902,A 0.000,B 0.000,C 90.000,E1 18.362} C_DIS
LIN {X -0.215,Y -446.364,Z 586.889,A 0.000,B 0.000,C 90.000,E1 16.079} C_DIS
LIN {X -0.005,Y -446.954,Z 586.880,A 0.000,B 0.000,C 90.000,E1 14.426} C_DIS
LIN {X -0.033,Y -447.788,Z 586.869,A 0.000,B 0.000,C 90.000,E1 12.479} C_DIS
LIN {X 0.108,Y -448.700,Z 586.860,A 0.000,B 0.000,C 90.000,E1 10.838} C_DIS
LIN {X -0.127,Y -450.279,Z 586.846,A 0.000,B 0.000,C 90.000,E1 8.276} C_DIS
LIN {X -0.061,Y -452.223,Z 586.832,A 0.000,B 0.000,C 90.000,E1 5.682} C_DIS
LIN {X 0.024,Y -454.547,Z 586.817,A 0.000,B 0.000,C 90.000,E1 3.094} C_DIS
LIN {X 0.013,Y -456.181,Z 586.808,A 0.000,B 0.000,C 90.000,E1 1.489} C_DIS
LIN {X -0.164,Y -459.336,Z 586.794,A 0.000,B 0.000,C 90.000,E1 358.854} C_DIS
LIN {X 0.097,Y -462.884,Z 586.779,A 0.000,B 0.000,C 90.000,E1 356.274} C_DIS
LIN {X 0.069,Y -465.627,Z 586.769,A 0.000,B 0.000,C 90.000,E1 354.375} C_DIS
LIN {X -0.093,Y -469.059,Z 586.757,A 0.000,B 0.000,C 90.000,E1 352.186} C_DIS
LIN {X -0.156,Y -471.466,Z 586.748,A 0.000,B 0.000,C 90.000,E1 350.622} C_DIS
LIN {X 0.034,Y -474.869,Z 586.736,A 0.000,B 0.000,C 90.000,E1 348.409} C_DIS
LIN {X -0.208,Y -477.417,Z 586.727,A 0.000,B 0.000,C 90.000,E1 346.881} C_DIS
LIN {X 0.181,Y -480.066,Z 586.718,A 0.000,B 0.000,C 90.000,E1 345.283} C_DIS
LIN {X 0.003,Y -484.689,Z 586.705,A 0.000,B 0.000,C 90.000,E1 342.834} C_DIS
LIN {X 0.102,Y -489.320,Z 586.691,A 0.000,B 0.000,C 90.000,E1 340.369} C_DIS
LIN {X 0.078,Y -492.265,Z 586.683,A 0.000,B 0.000,C 90.000,E1 338.847} C_DIS
LIN {X -0.126,Y -495.594,Z 586.672,A 0.000,B 0.000,C 90.000,E1 337.050} C_DIS
LIN {X -0.116,Y -498.188,Z 586.664,A 0.000,B 0.000,C 90.000,E1 335.537} C_DIS
LIN {X -0.117,Y -500.110,Z 586.657,A 0.000,B 0.000,C 90.000,E1 334.332} C_DIS
LIN {X -0.028,Y -502.537,Z 586.649,A 0.000,B 0.000,C 90.000,E1 332.820} C_DIS
LIN {X 0.053,Y -505.793,Z 586.637,A 0.000,B 0.000,C 90.000,E1 330.717} C_DIS
LIN {X 0.118,Y -509.547,Z 586.624,A 0.000,B 0.000,C 90.000,E1 328.329} C_DIS
LIN {X 0.230,Y -512.003,Z 586.616,A 0.000,B 0.000,C 90.000,E1 326.834} C_DIS
LIN {X 0.231,Y -515.647,Z 586.604,A 0.000,B 0.000,C 90.000,E1 324.769} C_DIS
LIN {X -0.221,Y -519.451,Z 586.593,A 0.000,B 0.000,C 90.000,E1 322.763} C_DIS
LIN {X -0.302,Y -523.896,Z 586.580,A 0.000,B 0.000,C 90.000,E1 320.436} C_DIS
LIN {X 0.130,Y -527.516,Z 586.570,A 0.000,B 0.000,C 90.000,E1 318.647} C_DIS
LIN {X -0.021,Y -529.903,Z 586.566,A 0.000,B 0.000,C 90.000,E1 317.796} C_DIS
LIN {X 0.005,Y -532.716,Z 586.561,A 0.000,B 0.000,C 90.000,E1 316.944} C_DIS
LIN {X -0.045,Y -534.157,Z 586.559,A 0.000,B 0.000,C 90.000,E1 316.662} C_DIS
LIN {X 0.235,Y -536.555,Z 586.557,A 0.000,B 0.000,C 90.000,E1 316.215} C_DIS
LIN {X -0.042,Y -539.832,Z 586.555,A 0.000,B 0.000,C 90.000,E1 315.810} C_DIS
LIN {X 0.233,Y -544.175,Z 586.552,A 0.000,B 0.000,C 90.000,E1 315.324} C_DIS
LIN {X -0.300,Y -548.366,Z 586.550,A 0.000,B 0.000,C 90.000,E1 315.000} C_DIS
LIN {X 0.041,Y -554.470,Z 586.547,A 0.000,B 0.000,C 90.000,E1 314.474} C_DIS
LIN {X 0.199,Y -568.990,Z 586.541,A 0.000,B 0.000,C 90.000,E1 313.380} C_DIS
LIN {X -0.386,Y -579.233,Z 586.537,A 0.000,B 0.000,C 90.000,E1 312.690} C_DIS
LIN {X 0.020,Y -589.377,Z 586.533,A 0.000,B 0.000,C 90.000,E1 311.919} C_DIS
LIN {X 0.105,Y -596.333,Z 586.530,A 0.000,B 0.000,C 90.000,E1 311.391} C_DIS
LIN {X 0.073,Y -600.453,Z 586.528,A 0.000,B 0.000,C 90.000,E1 311.067} C_DIS
LIN {X -0.173,Y -603.246,Z 586.527,A 0.000,B 0.000,C 90.000,E1 310.862} C_DIS
LIN {X 0.241,Y -608.253,Z 586.524,A 0.000,B 0.000,C 90.000,E1 310.378} C_DIS
LIN {X 0.332,Y -612.097,Z 586.523,A 0.000,B 0.000,C 90.000,E1 310.011} C_DIS
LIN {X -0.128,Y -617.021,Z 586.520,A 0.000,B 0.000,C 90.000,E1 309.564} C_DIS
LIN {X 0.103,Y -621.763,Z 586.517,A 0.000,B 0.000,C 90.000,E1 309.036} C_DIS
LIN {X -0.231,Y -628.603,Z 586.513,A 0.000,B 0.000,C 90.000,E1 308.302} C_DIS
LIN {X -0.128,Y -636.883,Z 586.507,A 0.000,B 0.000,C 90.000,E1 307.282} C_DIS
LIN {X -0.227,Y -640.786,Z 586.504,A 0.000,B 0.000,C 90.000,E1 306.790} C_DIS
LIN {X 0.114,Y -647.114,Z 586.499,A 0.000,B 0.000,C 90.000,E1 305.884} C_DIS
LIN {X -0.027,Y -652.000,Z 586.495,A 0.000,B 0.000,C 90.000,E1 305.152} C_DIS
LIN {X 0.080,Y -654.323,Z 586.493,A 0.000,B 0.000,C 90.000,E1 304.771} C_DIS
LIN {X -0.002,Y -658.426,Z 586.489,A 0.000,B 0.000,C 90.000,E1 304.040} C_DIS
LIN {X 0.071,Y -661.470,Z 586.486,A 0.000,B 0.000,C 90.000,E1 303.420} C_DIS
LIN {X 0.228,Y -664.805,Z 586.482,A 0.000,B 0.000,C 90.000,E1 302.673} C_DIS
LIN {X 0.065,Y -667.940,Z 586.478,A 0.000,B 0.000,C 90.000,E1 301.957} C_DIS
LIN {X 0.036,Y -672.903,Z 586.471,A 0.000,B 0.000,C 90.000,E1 300.747} C_DIS
LIN {X -0.102,Y -676.679,Z 586.466,A 0.000,B 0.000,C 90.000,E1 299.795} C_DIS
LIN {X 0.056,Y -680.158,Z 586.460,A 0.000,B 0.000,C 90.000,E1 298.821} C_DIS
LIN {X 0.058,Y -682.541,Z 586.456,A 0.000,B 0.000,C 90.000,E1 298.103} C_DIS
LIN {X 0.297,Y -685.518,Z 586.451,A 0.000,B 0.000,C 90.000,E1 297.129} C_DIS
LIN {X 0.038,Y -687.406,Z 586.447,A 0.000,B 0.000,C 90.000,E1 296.437} C_DIS
LIN {X -0.353,Y -687.762,Z 586.446,A 0.000,B 0.000,C 90.000,E1 296.232} C_DIS
LIN {X 0.102,Y -688.034,Z 586.443,A 0.000,B 0.000,C 90.000,E1 295.720} C_DIS
LIN {X 0.329,Y -687.770,Z 586.442,A 0.000,B 0.000,C 90.000,E1 295.463} C_DIS
LIN {X -0.131,Y -686.091,Z 586.439,A 0.000,B 0.000,C 90.000,E1 295.027} C_DIS
LIN {X -0.019,Y -685.578,Z 586.438,A 0.000,B 0.000,C 90.000,E1 294.899} C_DIS
LIN {X 0.092,Y -684.732,Z 586.438,A 0.000,B 0.000,C 90.000,E1 294.771} C_DIS
LIN {X -0.403,Y -680.900,Z 586.436,A 0.000,B 0.000,C 90.000,E1 294.463} C_DIS
LIN {X -0.212,Y -679.807,Z 586.435,A 0.000,B 0.000,C 90.000,E1 294.335} C_DIS
LIN {X -0.035,Y -678.271,Z 586.435,A 0.000,B 0.000,C 90.000,E1 294.207} C_DIS
LIN {X 0.141,Y -675.631,Z 586.434,A 0.000,B 0.000,C 90.000,E1 294.079} C_DIS
LIN {X -0.012,Y -672.023,Z 586.433,A 0.000,B 0.000,C 90.000,E1 293.951} C_DIS
LIN {X 0.361,Y -669.793,Z 586.433,A 0.000,B 0.000,C 90.000,E1 293.823} C_DIS
LIN {X 0.144,Y -667.377,Z 586.432,A 0.000,B 0.000,C 90.000,E1 293.770} C_DIS
LIN {X 0.197,Y -664.315,Z 586.432,A 0.000,B 0.000,C 90.000,E1 293.695} C_DIS
LIN {X 0.111,Y -662.138,Z 586.431,A 0.000,B 0.000,C 90.000,E1 293.643} C_DIS
LIN {X -0.206,Y -639.131,Z 586.429,A 0.000,B 0.000,C 90.000,E1 293.259} C_DIS
LIN {X 0.074,Y -629.757,Z 586.428,A 0.000,B 0.000,C 90.000,E1 293.025} C_DIS
LIN {X -0.094,Y -616.380,Z 586.426,A 0.000,B 0.000,C 90.000,E1 292.695} C_DIS
LIN {X 0.081,Y -602.973,Z 586.424,A 0.000,B 0.000,C 90.000,E1 292.280} C_DIS
LIN {X -0.240,Y -580.400,Z 586.420,A 0.000,B 0.000,C 90.000,E1 291.589} C_DIS
LIN {X 0.144,Y -571.680,Z 586.418,A 0.000,B 0.000,C 90.000,E1 291.280} C_DIS
LIN {X -0.224,Y -566.472,Z 586.417,A 0.000,B 0.000,C 90.000,E1 291.099} C_DIS
LIN {X 0.212,Y -561.935,Z 586.416,A 0.000,B 0.000,C 90.000,E1 290.791} C_DIS
LIN {X 0.183,Y -561.915,Z 586.416,A 0.000,B 0.000,C 90.000,E1 290.791} C_DIS
LIN {X -0.223,Y -560.964,Z 586.415,A 0.000,B 0.000,C 90.000,E1 290.663} C_DIS
LIN {X 0.169,Y -560.409,Z 586.412,A 0.000,B 0.000,C 90.000,E1 290.174} C_DIS
LIN {X -0.135,Y -560.460,Z 586.405,A 0.000,B 0.000,C 90.000,E1 288.833} C_DIS
LIN {X 0.196,Y -560.253,Z 586.398,A 0.000,B 0.000,C 90.000,E1 287.692} C_DIS
LIN {X -0.139,Y -559.553,Z 586.388,A 0.000,B 0.000,C 90.000,E1 285.788} C_DIS
LIN {X -0.088,Y -558.677,Z 586.378,A 0.000,B 0.000,C 90.000,E1 284.120} C_DIS
LIN {X -0.207,Y -557.736,Z 586.369,A 0.000,B 0.000,C 90.000,E1 282.467} C_DIS
LIN {X 0.104,Y -556.638,Z 586.358,A 0.000,B 0.000,C 90.000,E1 280.489} C_DIS
LIN {X 0.137,Y -555.826,Z 586.351,A 0.000,B 0.000,C 90.000,E1 279.095} C_DIS
LIN {X 0.151,Y -555.132,Z 586.343,A 0.000,B 0.000,C 90.000,E1 277.701} C_DIS
LIN {X 0.130,Y -554.331,Z 586.334,A 0.000,B 0.000,C 90.000,E1 276.030} C_DIS
LIN {X -0.166,Y -553.396,Z 586.318,A 0.000,B 0.000,C 90.000,E1 273.269} C_DIS
LIN {X -0.211,Y -552.888,Z 586.307,A 0.000,B 0.000,C 90.000,E1 271.318} C_DIS
LIN {X 0.119,Y -552.445,Z 586.299,A 0.000,B 0.000,C 90.000,E1 269.885} C_DIS
LIN {X 0.028,Y -551.691,Z 586.289,A 0.000,B 0.000,C 90.000,E1 267.936} C_DIS
LIN {X -0.091,Y -550.891,Z 586.278,A 0.000,B 0.000,C 90.000,E1 265.988} C_DIS
LIN {X 0.240,Y -550.163,Z 586.270,A 0.000,B 0.000,C 90.000,E1 264.552} C_DIS
LIN {X 0.069,Y -549.319,Z 586.262,A 0.000,B 0.000,C 90.000,E1 263.166} C_DIS
LIN {X -0.141,Y -548.450,Z 586.256,A 0.000,B 0.000,C 90.000,E1 262.064} C_DIS
LIN {X -0.144,Y -546.517,Z 586.245,A 0.000,B 0.000,C 90.000,E1 260.095} C_DIS
LIN {X -0.210,Y -544.883,Z 586.236,A 0.000,B 0.000,C 90.000,E1 258.409} C_DIS
LIN {X -0.176,Y -543.453,Z 586.228,A 0.000,B 0.000,C 90.000,E1 256.992} C_DIS
LIN {X 0.068,Y -541.122,Z 586.215,A 0.000,B 0.000,C 90.000,E1 254.700} C_DIS
LIN {X -0.126,Y -539.321,Z 586.206,A 0.000,B 0.000,C 90.000,E1 253.015} C_DIS
LIN {X -0.096,Y -538.041,Z 586.199,A 0.000,B 0.000,C 90.000,E1 251.873} C_DIS
LIN {X -0.089,Y -536.557,Z 586.193,A 0.000,B 0.000,C 90.000,E1 250.732} C_DIS
LIN {X -0.140,Y -535.261,Z 586.188,A 0.000,B 0.000,C 90.000,E1 249.880} C_DIS
LIN {X -0.003,Y -533.333,Z 586.182,A 0.000,B 0.000,C 90.000,E1 248.720} C_DIS
LIN {X 0.104,Y -531.754,Z 586.177,A 0.000,B 0.000,C 90.000,E1 247.847} C_DIS
LIN {X -0.100,Y -529.472,Z 586.171,A 0.000,B 0.000,C 90.000,E1 246.719} C_DIS
LIN {X 0.018,Y -525.927,Z 586.161,A 0.000,B 0.000,C 90.000,E1 244.973} C_DIS
LIN {X 0.110,Y -522.753,Z 586.153,A 0.000,B 0.000,C 90.000,E1 243.512} C_DIS
LIN {X -0.083,Y -519.408,Z 586.145,A 0.000,B 0.000,C 90.000,E1 242.076} C_DIS
LIN {X -0.280,Y -518.064,Z 586.142,A 0.000,B 0.000,C 90.000,E1 241.513} C_DIS
LIN {X -0.218,Y -515.050,Z 586.135,A 0.000,B 0.000,C 90.000,E1 240.333} C_DIS
LIN {X 0.048,Y -510.408,Z 586.125,A 0.000,B 0.000,C 90.000,E1 238.535} C_DIS
LIN {X 0.150,Y -506.584,Z 586.117,A 0.000,B 0.000,C 90.000,E1 237.041} C_DIS
LIN {X -0.131,Y -503.279,Z 586.110,A 0.000,B 0.000,C 90.000,E1 235.881} C_DIS
LIN {X -0.059,Y -500.683,Z 586.105,A 0.000,B 0.000,C 90.000,E1 234.975} C_DIS
LIN {X -0.272,Y -492.434,Z 586.089,A 0.000,B 0.000,C 90.000,E1 231.984} C_DIS
LIN {X -0.086,Y -485.186,Z 586.073,A 0.000,B 0.000,C 90.000,E1 229.218} C_DIS
LIN {X 0.014,Y -478.983,Z 586.060,A 0.000,B 0.000,C 90.000,E1 226.743} C_DIS
LIN {X 0.033,Y -474.458,Z 586.049,A 0.000,B 0.000,C 90.000,E1 224.879} C_DIS
LIN {X 0.185,Y -470.781,Z 586.041,A 0.000,B 0.000,C 90.000,E1 223.299} C_DIS
LIN {X -0.220,Y -465.776,Z 586.029,A 0.000,B 0.000,C 90.000,E1 221.148} C_DIS
LIN {X -0.045,Y -461.009,Z 586.016,A 0.000,B 0.000,C 90.000,E1 218.910} C_DIS
LIN {X -0.040,Y -457.715,Z 586.007,A 0.000,B 0.000,C 90.000,E1 217.317} C_DIS
LIN {X 0.065,Y -452.467,Z 585.993,A 0.000,B 0.000,C 90.000,E1 214.739} C_DIS
LIN {X -0.171,Y -448.700,Z 585.982,A 0.000,B 0.000,C 90.000,E1 212.832} C_DIS
LIN {X 0.021,Y -444.013,Z 585.968,A 0.000,B 0.000,C 90.000,E1 210.207} C_DIS
LIN {X 0.126,Y -440.491,Z 585.957,A 0.000,B 0.000,C 90.000,E1 208.231} C_DIS
LIN {X -0.094,Y -437.602,Z 585.948,A 0.000,B 0.000,C 90.000,E1 206.616} C_DIS
LIN {X -0.158,Y -434.163,Z 585.937,A 0.000,B 0.000,C 90.000,E1 204.643} C_DIS
LIN {X 0.103,Y -431.968,Z 585.929,A 0.000,B 0.000,C 90.000,E1 203.281} C_DIS
LIN {X -0.076,Y -428.245,Z 585.917,A 0.000,B 0.000,C 90.000,E1 200.972} C_DIS
LIN {X -0.089,Y -424.229,Z 585.902,A 0.000,B 0.000,C 90.000,E1 198.290} C_DIS
LIN {X -0.042,Y -420.134,Z 585.885,A 0.000,B 0.000,C 90.000,E1 195.245} C_DIS
LIN {X -0.007,Y -418.343,Z 585.877,A 0.000,B 0.000,C 90.000,E1 193.883} C_DIS
LIN {X -0.098,Y -416.374,Z 585.870,A 0.000,B 0.000,C 90.000,E1 192.535} C_DIS
LIN {X -0.170,Y -413.897,Z 585.860,A 0.000,B 0.000,C 90.000,E1 190.838} C_DIS
LIN {X 0.042,Y -411.650,Z 585.851,A 0.000,B 0.000,C 90.000,E1 189.095} C_DIS
LIN {X 0.202,Y -409.707,Z 585.841,A 0.000,B 0.000,C 90.000,E1 187.352} C_DIS
LIN {X -0.193,Y -407.579,Z 585.831,A 0.000,B 0.000,C 90.000,E1 185.682} C_DIS
LIN {X 0.180,Y -405.925,Z 585.824,A 0.000,B 0.000,C 90.000,E1 184.245} C_DIS
LIN {X 0.188,Y -401.454,Z 585.797,A 0.000,B 0.000,C 90.000,E1 179.370} C_DIS
LIN {X -0.109,Y -399.905,Z 585.783,A 0.000,B 0.000,C 90.000,E1 176.963} C_DIS
LIN {X -0.058,Y -398.586,Z 585.766,A 0.000,B 0.000,C 90.000,E1 173.799} C_DIS
LIN {X 0.062,Y -398.060,Z 585.750,A 0.000,B 0.000,C 90.000,E1 170.971} C_DIS
LIN {X -0.044,Y -397.908,Z 585.734,A 0.000,B 0.000,C 90.000,E1 168.173} C_DIS
LIN {X 0.043,Y -398.311,Z 585.721,A 0.000,B 0.000,C 90.000,E1 165.700} C_DIS
LIN {X -0.147,Y -398.900,Z 585.707,A 0.000,B 0.000,C 90.000,E1 163.268} C_DIS
LIN {X -0.050,Y -399.623,Z 585.695,A 0.000,B 0.000,C 90.000,E1 161.148} C_DIS
LIN {X 0.067,Y -400.475,Z 585.684,A 0.000,B 0.000,C 90.000,E1 159.028} C_DIS
LIN {X -0.177,Y -401.624,Z 585.670,A 0.000,B 0.000,C 90.000,E1 156.613} C_DIS
LIN {X 0.049,Y -402.647,Z 585.658,A 0.000,B 0.000,C 90.000,E1 154.485} C_DIS
LIN {X -0.071,Y -403.669,Z 585.647,A 0.000,B 0.000,C 90.000,E1 152.410} C_DIS
LIN {X 0.039,Y -404.334,Z 585.639,A 0.000,B 0.000,C 90.000,E1 151.001} C_DIS
LIN {X 0.010,Y -405.200,Z 585.627,A 0.000,B 0.000,C 90.000,E1 148.918} C_DIS
LIN {X 0.009,Y -405.819,Z 585.616,A 0.000,B 0.000,C 90.000,E1 146.834} C_DIS
LIN {X -0.107,Y -406.302,Z 585.604,A 0.000,B 0.000,C 90.000,E1 144.769} C_DIS
LIN {X 0.112,Y -406.665,Z 585.595,A 0.000,B 0.000,C 90.000,E1 143.004} C_DIS
LIN {X -0.025,Y -407.186,Z 585.581,A 0.000,B 0.000,C 90.000,E1 140.598} C_DIS
LIN {X -0.082,Y -407.606,Z 585.570,A 0.000,B 0.000,C 90.000,E1 138.528} C_DIS
LIN {X 0.030,Y -407.818,Z 585.560,A 0.000,B 0.000,C 90.000,E1 136.782} C_DIS
LIN {X -0.017,Y -407.992,Z 585.552,A 0.000,B 0.000,C 90.000,E1 135.405} C_DIS
LIN {X 0.053,Y -408.293,Z 585.539,A 0.000,B 0.000,C 90.000,E1 132.975} C_DIS
LIN {X 0.030,Y -408.412,Z 585.531,A 0.000,B 0.000,C 90.000,E1 131.595} C_DIS
LIN {X 0.008,Y -408.496,Z 585.523,A 0.000,B 0.000,C 90.000,E1 130.216} C_DIS
LIN {X -0.119,Y -408.348,Z 585.514,A 0.000,B 0.000,C 90.000,E1 128.463} C_DIS
LIN {X -0.091,Y -415.202,Z 585.500,A 0.000,B 0.000,C 90.000,E1 126.091} C_DIS
LIN {X 0.020,Y -416.875,Z 585.497,A 0.000,B 0.000,C 90.000,E1 125.391} C_DIS
LIN {X -0.052,Y -426.594,Z 585.476,A 0.000,B 0.000,C 90.000,E1 121.671} C_DIS
LIN {X -0.089,Y -430.660,Z 585.469,A 0.000,B 0.000,C 90.000,E1 120.335} C_DIS
LIN {X -0.126,Y -430.725,Z 585.469,A 0.000,B 0.000,C 90.000,E1 120.335} C_DIS
LIN {X -0.090,Y -438.063,Z 585.467,A 0.000,B 0.000,C 90.000,E1 120.001} C_DIS
LIN {X -0.152,Y -453.717,Z 585.463,A 0.000,B 0.000,C 90.000,E1 119.283} C_DIS
LIN {X -0.031,Y -465.695,Z 585.459,A 0.000,B 0.000,C 90.000,E1 118.693} C_DIS
LIN {X -0.033,Y -477.552,Z 585.456,A 0.000,B 0.000,C 90.000,E1 118.103} C_DIS
LIN {X -0.050,Y -482.624,Z 585.455,A 0.000,B 0.000,C 90.000,E1 117.847} C_DIS
LIN {X -0.036,Y -493.942,Z 585.451,A 0.000,B 0.000,C 90.000,E1 117.206} C_DIS
LIN {X -0.151,Y -502.027,Z 585.449,A 0.000,B 0.000,C 90.000,E1 116.744} C_DIS
LIN {X -0.244,Y -508.386,Z 585.446,A 0.000,B 0.000,C 90.000,E1 116.360} C_DIS
LIN {X -0.240,Y -516.356,Z 585.443,A 0.000,B 0.000,C 90.000,E1 115.848} C_DIS
LIN {X -0.099,Y -527.125,Z 585.439,A 0.000,B 0.000,C 90.000,E1 115.079} C_DIS
LIN {X 0.015,Y -534.573,Z 585.436,A 0.000,B 0.000,C 90.000,E1 114.515} C_DIS
LIN {X -0.286,Y -538.989,Z 585.434,A 0.000,B 0.000,C 90.000,E1 114.207} C_DIS
LIN {X -0.075,Y -546.152,Z 585.431,A 0.000,B 0.000,C 90.000,E1 113.590} C_DIS
LIN {X -0.013,Y -547.622,Z 585.430,A 0.000,B 0.000,C 90.000,E1 113.462} C_DIS
LIN {X 0.281,Y -552.813,Z 585.428,A 0.000,B 0.000,C 90.000,E1 112.950} C_DIS
LIN {X -0.117,Y -557.553,Z 585.425,A 0.000,B 0.000,C 90.000,E1 112.514} C_DIS
LIN {X 0.206,Y -563.706,Z 585.421,A 0.000,B 0.000,C 90.000,E1 111.770} C_DIS
LIN {X 0.219,Y -566.716,Z 585.419,A 0.000,B 0.000,C 90.000,E1 111.354} C_DIS
LIN {X 0.023,Y -568.754,Z 585.417,A 0.000,B 0.000,C 90.000,E1 111.099} C_DIS
LIN {X 0.272,Y -571.470,Z 585.415,A 0.000,B 0.000,C 90.000,E1 110.663} C_DIS
LIN {X -0.113,Y -573.145,Z 585.413,A 0.000,B 0.000,C 90.000,E1 110.429} C_DIS
LIN {X -0.199,Y -577.672,Z 585.409,A 0.000,B 0.000,C 90.000,E1 109.631} C_DIS
LIN {X 0.290,Y -581.224,Z 585.405,A 0.000,B 0.000,C 90.000,E1 108.906} C_DIS
LIN {X -0.076,Y -585.747,Z 585.400,A 0.000,B 0.000,C 90.000,E1 108.000} C_DIS
LIN {X -0.323,Y -589.237,Z 585.396,A 0.000,B 0.000,C 90.000,E1 107.221} C_DIS
LIN {X 0.149,Y -594.571,Z 585.388,A 0.000,B 0.000,C 90.000,E1 105.843} C_DIS
LIN {X -0.018,Y -597.473,Z 585.384,A 0.000,B 0.000,C 90.000,E1 105.064} C_DIS
LIN {X 0.011,Y -602.914,Z 585.375,A 0.000,B 0.000,C 90.000,E1 103.480} C_DIS
LIN {X 0.169,Y -608.386,Z 585.366,A 0.000,B 0.000,C 90.000,E1 101.895} C_DIS
LIN {X -0.170,Y -613.819,Z 585.358,A 0.000,B 0.000,C 90.000,E1 100.366} C_DIS
LIN {X -0.053,Y -617.343,Z 585.352,A 0.000,B 0.000,C 90.000,E1 99.321} C_DIS
LIN {X -0.261,Y -619.868,Z 585.348,A 0.000,B 0.000,C 90.000,E1 98.568} C_DIS
LIN {X -0.148,Y -623.188,Z 585.342,A 0.000,B 0.000,C 90.000,E1 97.530} C_DIS
LIN {X 0.092,Y -626.360,Z 585.336,A 0.000,B 0.000,C 90.000,E1 96.486} C_DIS
LIN {X 0.009,Y -629.921,Z 585.329,A 0.000,B 0.000,C 90.000,E1 95.220} C_DIS
LIN {X -0.148,Y -631.780,Z 585.325,A 0.000,B 0.000,C 90.000,E1 94.473} C_DIS
LIN {X 0.081,Y -633.949,Z 585.319,A 0.000,B 0.000,C 90.000,E1 93.440} C_DIS
LIN {X 0.085,Y -636.220,Z 585.312,A 0.000,B 0.000,C 90.000,E1 92.178} C_DIS
LIN {X -0.017,Y -637.368,Z 585.308,A 0.000,B 0.000,C 90.000,E1 91.432} C_DIS
LIN {X 0.266,Y -638.509,Z 585.302,A 0.000,B 0.000,C 90.000,E1 90.401} C_DIS
LIN {X 0.171,Y -639.140,Z 585.298,A 0.000,B 0.000,C 90.000,E1 89.656} C_DIS
LIN {X 0.081,Y -639.521,Z 585.294,A 0.000,B 0.000,C 90.000,E1 88.912} C_DIS
LIN {X 0.233,Y -639.647,Z 585.291,A 0.000,B 0.000,C 90.000,E1 88.396} C_DIS
LIN {X -0.078,Y -639.489,Z 585.286,A 0.000,B 0.000,C 90.000,E1 87.421} C_DIS
LIN {X -0.140,Y -639.145,Z 585.281,A 0.000,B 0.000,C 90.000,E1 86.674} C_DIS
LIN {X 0.186,Y -638.445,Z 585.276,A 0.000,B 0.000,C 90.000,E1 85.641} C_DIS
LIN {X -0.142,Y -637.366,Z 585.270,A 0.000,B 0.000,C 90.000,E1 84.666} C_DIS
LIN {X 0.206,Y -636.134,Z 585.265,A 0.000,B 0.000,C 90.000,E1 83.628} C_DIS
LIN {X -0.256,Y -635.381,Z 585.262,A 0.000,B 0.000,C 90.000,E1 83.166} C_DIS
LIN {X 0.062,Y -633.513,Z 585.256,A 0.000,B 0.000,C 90.000,E1 82.129} C_DIS
LIN {X 0.011,Y -631.936,Z 585.252,A 0.000,B 0.000,C 90.000,E1 81.376} C_DIS
LIN {X -0.252,Y -629.635,Z 585.247,A 0.000,B 0.000,C 90.000,E1 80.387} C_DIS
LIN {X 0.074,Y -627.067,Z 585.241,A 0.000,B 0.000,C 90.000,E1 79.342} C_DIS
LIN {X -0.130,Y -624.292,Z 585.235,A 0.000,B 0.000,C 90.000,E1 78.342} C_DIS
LIN {X 0.110,Y -621.369,Z 585.230,A 0.000,B 0.000,C 90.000,E1 77.297} C_DIS
LIN {X 0.355,Y -617.281,Z 585.222,A 0.000,B 0.000,C 90.000,E1 75.992} C_DIS
LIN {X 0.260,Y -614.609,Z 585.218,A 0.000,B 0.000,C 90.000,E1 75.227} C_DIS
LIN {X 0.133,Y -611.710,Z 585.214,A 0.000,B 0.000,C 90.000,E1 74.464} C_DIS
LIN {X -0.193,Y -609.645,Z 585.211,A 0.000,B 0.000,C 90.000,E1 73.976} C_DIS
LIN {X -0.200,Y -606.313,Z 585.207,A 0.000,B 0.000,C 90.000,E1 73.196} C_DIS
LIN {X -0.194,Y -603.351,Z 585.203,A 0.000,B 0.000,C 90.000,E1 72.543} C_DIS
LIN {X -0.272,Y -599.534,Z 585.199,A 0.000,B 0.000,C 90.000,E1 71.764} C_DIS
LIN {X 0.309,Y -594.651,Z 585.193,A 0.000,B 0.000,C 90.000,E1 70.786} C_DIS
LIN {X 0.132,Y -590.091,Z 585.189,A 0.000,B 0.000,C 90.000,E1 70.007} C_DIS
LIN {X 0.170,Y -585.886,Z 585.185,A 0.000,B 0.000,C 90.000,E1 69.337} C_DIS
LIN {X -0.093,Y -581.445,Z 585.182,A 0.000,B 0.000,C 90.000,E1 68.720} C_DIS
LIN {X 0.085,Y -576.360,Z 585.178,A 0.000,B 0.000,C 90.000,E1 68.028} C_DIS
LIN {X 0.085,Y -571.914,Z 585.175,A 0.000,B 0.000,C 90.000,E1 67.486} C_DIS
LIN {X -0.218,Y -567.156,Z 585.172,A 0.000,B 0.000,C 90.000,E1 66.975} C_DIS
LIN {X -0.125,Y -562.074,Z 585.169,A 0.000,B 0.000,C 90.000,E1 66.433} C_DIS
LIN {X 0.191,Y -557.066,Z 585.166,A 0.000,B 0.000,C 90.000,E1 65.921} C_DIS
LIN {X -0.179,Y -551.516,Z 585.164,A 0.000,B 0.000,C 90.000,E1 65.485} C_DIS
LIN {X 0.171,Y -547.092,Z 585.162,A 0.000,B 0.000,C 90.000,E1 65.101} C_DIS
LIN {X -0.206,Y -540.992,Z 585.159,A 0.000,B 0.000,C 90.000,E1 64.717} C_DIS
LIN {X -0.258,Y -535.906,Z 585.158,A 0.000,B 0.000,C 90.000,E1 64.409} C_DIS
LIN {X -0.162,Y -529.133,Z 585.156,A 0.000,B 0.000,C 90.000,E1 64.024} C_DIS
LIN {X 0.291,Y -522.378,Z 585.154,A 0.000,B 0.000,C 90.000,E1 63.640} C_DIS
LIN {X 0.159,Y -515.412,Z 585.152,A 0.000,B 0.000,C 90.000,E1 63.332} C_DIS
LIN {X 0.223,Y -504.997,Z 585.149,A 0.000,B 0.000,C 90.000,E1 62.871} C_DIS
LIN {X -0.154,Y -493.020,Z 585.147,A 0.000,B 0.000,C 90.000,E1 62.410} C_DIS
LIN {X -0.268,Y -459.027,Z 585.138,A 0.000,B 0.000,C 90.000,E1 60.923} C_DIS
LIN {X 0.091,Y -452.272,Z 585.136,A 0.000,B 0.000,C 90.000,E1 60.539} C_DIS
LIN {X 0.049,Y -452.171,Z 585.136,A 0.000,B 0.000,C 90.000,E1 60.539} C_DIS
LIN {X -0.028,Y -443.952,Z 585.114,A 0.000,B 0.000,C 90.000,E1 56.501} C_DIS
LIN {X -0.001,Y -434.547,Z 585.091,A 0.000,B 0.000,C 90.000,E1 52.431} C_DIS
LIN {X -0.084,Y -434.969,Z 585.088,A 0.000,B 0.000,C 90.000,E1 51.904} C_DIS
LIN {X -0.010,Y -436.847,Z 585.077,A 0.000,B 0.000,C 90.000,E1 49.908} C_DIS
LIN {X 0.061,Y -438.714,Z 585.066,A 0.000,B 0.000,C 90.000,E1 47.919} C_DIS
LIN {X -0.152,Y -440.566,Z 585.055,A 0.000,B 0.000,C 90.000,E1 45.972} C_DIS
LIN {X 0.031,Y -441.759,Z 585.048,A 0.000,B 0.000,C 90.000,E1 44.636} C_DIS
LIN {X -0.069,Y -442.777,Z 585.041,A 0.000,B 0.000,C 90.000,E1 43.338} C_DIS
LIN {X 0.132,Y -443.735,Z 585.032,A 0.000,B 0.000,C 90.000,E1 41.676} C_DIS
LIN {X 0.070,Y -444.344,Z 585.024,A 0.000,B 0.000,C 90.000,E1 40.378} C_DIS
LIN {X 0.074,Y -444.876,Z 585.017,A 0.000,B 0.000,C 90.000,E1 39.072} C_DIS
LIN {X -0.257,Y -445.261,Z 585.010,A 0.000,B 0.000,C 90.000,E1 37.810} C_DIS
LIN {X 0.070,Y -445.480,Z 585.005,A 0.000,B 0.000,C 90.000,E1 36.790} C_DIS
LIN {X -0.116,Y -445.596,Z 584.995,A 0.000,B 0.000,C 90.000,E1 35.185} C_DIS
LIN {X 0.012,Y -445.569,Z 584.988,A 0.000,B 0.000,C 90.000,E1 33.865} C_DIS
LIN {X -0.117,Y -445.432,Z 584.977,A 0.000,B 0.000,C 90.000,E1 31.926} C_DIS
LIN {X 0.039,Y -445.378,Z 584.966,A 0.000,B 0.000,C 90.000,E1 29.951} C_DIS
LIN {X 0.140,Y -445.329,Z 584.957,A 0.000,B 0.000,C 90.000,E1 28.309} C_DIS
LIN {X 0.029,Y -445.353,Z 584.948,A 0.000,B 0.000,C 90.000,E1 26.693} C_DIS
LIN {X 0.220,Y -445.375,Z 584.936,A 0.000,B 0.000,C 90.000,E1 24.387} C_DIS
LIN {X 0.126,Y -445.560,Z 584.927,A 0.000,B 0.000,C 90.000,E1 22.770} C_DIS
LIN {X -0.101,Y -445.764,Z 584.916,A 0.000,B 0.000,C 90.000,E1 20.844} C_DIS
LIN {X 0.061,Y -446.126,Z 584.903,A 0.000,B 0.000,C 90.000,E1 18.544} C_DIS
LIN {X 0.102,Y -446.619,Z 584.890,A 0.000,B 0.000,C 90.000,E1 16.260} C_DIS
LIN {X 0.171,Y -447.291,Z 584.880,A 0.000,B 0.000,C 90.000,E1 14.300} C_DIS
LIN {X 0.142,Y -448.097,Z 584.869,A 0.000,B 0.000,C 90.000,E1 12.355} C_DIS
LIN {X -0.242,Y -448.983,Z 584.860,A 0.000,B 0.000,C 90.000,E1 10.782} C_DIS
LIN {X -0.216,Y -450.357,Z 584.847,A 0.000,B 0.000,C 90.000,E1 8.511} C_DIS
LIN {X -0.094,Y -452.233,Z 584.833,A 0.000,B 0.000,C 90.000,E1 5.910} C_DIS
LIN {X -0.211,Y -454.194,Z 584.820,A 0.000,B 0.000,C 90.000,E1 3.669} C_DIS
LIN {X -0.029,Y -456.125,Z 584.810,A 0.000,B 0.000,C 90.000,E1 1.718} C_DIS
LIN {X -0.162,Y -459.474,Z 584.794,A 0.000,B 0.000,C 90.000,E1 358.854} C_DIS
LIN {X 0.103,Y -462.989,Z 584.779,A 0.000,B 0.000,C 90.000,E1 356.274} C_DIS
LIN {X -0.176,Y -465.262,Z 584.771,A 0.000,B 0.000,C 90.000,E1 354.723} C_DIS
LIN {X 0.171,Y -468.635,Z 584.758,A 0.000,B 0.000,C 90.000,E1 352.470} C_DIS
LIN {X -0.144,Y -471.566,Z 584.748,A 0.000,B 0.000,C 90.000,E1 350.622} C_DIS
LIN {X 0.049,Y -474.957,Z 584.736,A 0.000,B 0.000,C 90.000,E1 348.409} C_DIS
LIN {X 0.116,Y -477.979,Z 584.725,A 0.000,B 0.000,C 90.000,E1 346.533} C_DIS
LIN {X 0.199,Y -480.130,Z 584.718,A 0.000,B 0.000,C 90.000,E1 345.283} C_DIS
LIN {X 0.023,Y -484.707,Z 584.705,A 0.000,B 0.000,C 90.000,E1 342.834} C_DIS
LIN {X 0.122,Y -489.350,Z 584.691,A 0.000,B 0.000,C 90.000,E1 340.369} C_DIS
LIN {X 0.099,Y -492.294,Z 584.683,A 0.000,B 0.000,C 90.000,E1 338.847} C_DIS
LIN {X -0.105,Y -495.654,Z 584.672,A 0.000,B 0.000,C 90.000,E1 337.050} C_DIS
LIN {X -0.093,Y -498.249,Z 584.664,A 0.000,B 0.000,C 90.000,E1 335.537} C_DIS
LIN {X -0.093,Y -500.192,Z 584.657,A 0.000,B 0.000,C 90.000,E1 334.332} C_DIS
LIN {X -0.003,Y -502.627,Z 584.649,A 0.000,B 0.000,C 90.000,E1 332.820} C_DIS
LIN {X 0.081,Y -505.884,Z 584.637,A 0.000,B 0.000,C 90.000,E1 330.717} C_DIS
LIN {X 0.149,Y -509.668,Z 584.624,A 0.000,B 0.000,C 90.000,E1 328.329} C_DIS
LIN {X 0.263,Y -512.118,Z 584.616,A 0.000,B 0.000,C 90.000,E1 326.834} C_DIS
LIN {X -0.154,Y -515.761,Z 584.604,A 0.000,B 0.000,C 90.000,E1 324.815} C_DIS
LIN {X -0.123,Y -518.953,Z 584.595,A 0.000,B 0.000,C 90.000,E1 323.050} C_DIS
LIN {X -0.169,Y -522.812,Z 584.583,A 0.000,B 0.000,C 90.000,E1 321.009} C_DIS
LIN {X -0.259,Y -528.193,Z 584.569,A 0.000,B 0.000,C 90.000,E1 318.405} C_DIS
LIN {X -0.074,Y -531.390,Z 584.562,A 0.000,B 0.000,C 90.000,E1 317.229} C_DIS
LIN {X 0.232,Y -533.288,Z 584.559,A 0.000,B 0.000,C 90.000,E1 316.620} C_DIS
LIN {X 0.295,Y -535.072,Z 584.557,A 0.000,B 0.000,C 90.000,E1 316.296} C_DIS
LIN {X -0.078,Y -536.367,Z 584.556,A 0.000,B 0.000,C 90.000,E1 316.053} C_DIS
LIN {X 0.228,Y -539.369,Z 584.553,A 0.000,B 0.000,C 90.000,E1 315.567} C_DIS
LIN {X 0.069,Y -543.322,Z 584.551,A 0.000,B 0.000,C 90.000,E1 315.121} C_DIS
LIN {X 0.087,Y -547.090,Z 584.549,A 0.000,B 0.000,C 90.000,E1 314.757} C_DIS
LIN {X -0.006,Y -554.101,Z 584.546,A 0.000,B 0.000,C 90.000,E1 314.190} C_DIS
LIN {X -0.013,Y -574.871,Z 584.537,A 0.000,B 0.000,C 90.000,E1 312.651} C_DIS
LIN {X 0.056,Y -583.669,Z 584.533,A 0.000,B 0.000,C 90.000,E1 312.000} C_DIS
LIN {X 0.142,Y -592.152,Z 584.530,A 0.000,B 0.000,C 90.000,E1 311.391} C_DIS
LIN {X -0.124,Y -597.801,Z 584.528,A 0.000,B 0.000,C 90.000,E1 310.987} C_DIS
LIN {X 0.225,Y -601.928,Z 584.526,A 0.000,B 0.000,C 90.000,E1 310.620} C_DIS
LIN {X -0.040,Y -606.020,Z 584.524,A 0.000,B 0.000,C 90.000,E1 310.297} C_DIS
LIN {X -0.170,Y -612.295,Z 584.521,A 0.000,B 0.000,C 90.000,E1 309.725} C_DIS
LIN {X -0.193,Y -616.048,Z 584.519,A 0.000,B 0.000,C 90.000,E1 309.358} C_DIS
LIN {X 0.026,Y -620.809,Z 584.516,A 0.000,B 0.000,C 90.000,E1 308.830} C_DIS
LIN {X -0.354,Y -627.709,Z 584.512,A 0.000,B 0.000,C 90.000,E1 308.096} C_DIS
LIN {X 0.206,Y -635.092,Z 584.507,A 0.000,B 0.000,C 90.000,E1 307.156} C_DIS
LIN {X 0.086,Y -640.011,Z 584.503,A 0.000,B 0.000,C 90.000,E1 306.537} C_DIS
LIN {X -0.134,Y -644.598,Z 584.500,A 0.000,B 0.000,C 90.000,E1 305.931} C_DIS
LIN {X -0.149,Y -649.777,Z 584.495,A 0.000,B 0.000,C 90.000,E1 305.185} C_DIS
LIN {X 0.268,Y -654.365,Z 584.491,A 0.000,B 0.000,C 90.000,E1 304.405} C_DIS
LIN {X 0.267,Y -657.168,Z 584.489,A 0.000,B 0.000,C 90.000,E1 303.913} C_DIS
LIN {X -0.084,Y -659.676,Z 584.486,A 0.000,B 0.000,C 90.000,E1 303.452} C_DIS
LIN {X -0.018,Y -664.178,Z 584.480,A 0.000,B 0.000,C 90.000,E1 302.467} C_DIS
LIN {X 0.307,Y -668.362,Z 584.475,A 0.000,B 0.000,C 90.000,E1 301.465} C_DIS
LIN {X 0.276,Y -673.317,Z 584.468,A 0.000,B 0.000,C 90.000,E1 300.256} C_DIS
LIN {X -0.201,Y -676.997,Z 584.463,A 0.000,B 0.000,C 90.000,E1 299.333} C_DIS
LIN {X -0.233,Y -679.555,Z 584.459,A 0.000,B 0.000,C 90.000,E1 298.615} C_DIS
LIN {X -0.037,Y -682.649,Z 584.454,A 0.000,B 0.000,C 90.000,E1 297.641} C_DIS
LIN {X -0.018,Y -684.857,Z 584.450,A 0.000,B 0.000,C 90.000,E1 296.924} C_DIS
LIN {X 0.109,Y -686.090,Z 584.447,A 0.000,B 0.000,C 90.000,E1 296.437} C_DIS
LIN {X -0.286,Y -686.476,Z 584.446,A 0.000,B 0.000,C 90.000,E1 296.232} C_DIS
LIN {X 0.159,Y -686.790,Z 584.443,A 0.000,B 0.000,C 90.000,E1 295.720} C_DIS
LIN {X 0.383,Y -686.438,Z 584.442,A 0.000,B 0.000,C 90.000,E1 295.463} C_DIS
LIN {X -0.308,Y -685.756,Z 584.440,A 0.000,B 0.000,C 90.000,E1 295.283} C_DIS
LIN {X -0.085,Y -684.913,Z 584.439,A 0.000,B 0.000,C 90.000,E1 295.027} C_DIS
LIN {X 0.025,Y -684.309,Z 584.438,A 0.000,B 0.000,C 90.000,E1 294.899} C_DIS
LIN {X 0.134,Y -683.336,Z 584.438,A 0.000,B 0.000,C 90.000,E1 294.771} C_DIS
LIN {X 0.347,Y -680.755,Z 584.436,A 0.000,B 0.000,C 90.000,E1 294.515} C_DIS
LIN {X 0.002,Y -679.337,Z 584.436,A 0.000,B 0.000,C 90.000,E1 294.387} C_DIS
LIN {X 0.101,Y -677.920,Z 584.435,A 0.000,B 0.000,C 90.000,E1 294.259} C_DIS
LIN {X -0.077,Y -675.478,Z 584.434,A 0.000,B 0.000,C 90.000,E1 294.155} C_DIS
LIN {X 0.213,Y -668.269,Z 584.432,A 0.000,B 0.000,C 90.000,E1 293.823} C_DIS
LIN {X 0.122,Y -663.426,Z 584.432,A 0.000,B 0.000,C 90.000,E1 293.695} C_DIS
LIN {X 0.187,Y -658.580,Z 584.431,A 0.000,B 0.000,C 90.000,E1 293.590} C_DIS
LIN {X 0.159,Y -637.932,Z 584.429,A 0.000,B 0.000,C 90.000,E1 293.206} C_DIS
LIN {X 0.158,Y -624.658,Z 584.427,A 0.000,B 0.000,C 90.000,E1 292.898} C_DIS
LIN {X 0.336,Y -611.200,Z 584.425,A 0.000,B 0.000,C 90.000,E1 292.514} C_DIS
LIN {X -0.231,Y -578.559,Z 584.420,A 0.000,B 0.000,C 90.000,E1 291.535} C_DIS
LIN {X -0.046,Y -573.164,Z 584.419,A 0.000,B 0.000,C 90.000,E1 291.354} C_DIS
LIN {X 0.229,Y -566.330,Z 584.417,A 0.000,B 0.000,C 90.000,E1 291.046} C_DIS
LIN {X 0.201,Y -562.168,Z 584.416,A 0.000,B 0.000,C 90.000,E1 290.791} C_DIS
LIN {X 0.173,Y -562.120,Z 584.416,A 0.000,B 0.000,C 90.000,E1 290.791} C_DIS
LIN {X -0.171,Y -561.281,Z 584.415,A 0.000,B 0.000,C 90.000,E1 290.663} C_DIS
LIN {X -0.116,Y -560.699,Z 584.412,A 0.000,B 0.000,C 90.000,E1 290.174} C_DIS
LIN {X 0.114,Y -560.813,Z 584.404,A 0.000,B 0.000,C 90.000,E1 288.779} C_DIS
LIN {X -0.080,Y -560.578,Z 584.398,A 0.000,B 0.000,C 90.000,E1 287.692} C_DIS
LIN {X -0.147,Y -560.069,Z 584.391,A 0.000,B 0.000,C 90.000,E1 286.315} C_DIS
LIN {X -0.115,Y -559.732,Z 584.386,A 0.000,B 0.000,C 90.000,E1 285.481} C_DIS
LIN {X -0.206,Y -558.845,Z 584.377,A 0.000,B 0.000,C 90.000,E1 283.828} C_DIS
LIN {X 0.084,Y -558.029,Z 584.369,A 0.000,B 0.000,C 90.000,E1 282.411} C_DIS
LIN {X -0.280,Y -557.101,Z 584.360,A 0.000,B 0.000,C 90.000,E1 280.782} C_DIS
LIN {X -0.146,Y -556.305,Z 584.352,A 0.000,B 0.000,C 90.000,E1 279.378} C_DIS
LIN {X -0.082,Y -555.439,Z 584.343,A 0.000,B 0.000,C 90.000,E1 277.701} C_DIS
LIN {X -0.155,Y -554.787,Z 584.335,A 0.000,B 0.000,C 90.000,E1 276.315} C_DIS
LIN {X -0.061,Y -553.943,Z 584.323,A 0.000,B 0.000,C 90.000,E1 274.073} C_DIS
LIN {X -0.217,Y -553.564,Z 584.315,A 0.000,B 0.000,C 90.000,E1 272.694} C_DIS
LIN {X 0.137,Y -553.202,Z 584.307,A 0.000,B 0.000,C 90.000,E1 271.260} C_DIS
LIN {X -0.080,Y -552.751,Z 584.299,A 0.000,B 0.000,C 90.000,E1 269.885} C_DIS
LIN {X -0.245,Y -552.089,Z 584.290,A 0.000,B 0.000,C 90.000,E1 268.224} C_DIS
LIN {X 0.221,Y -551.287,Z 584.279,A 0.000,B 0.000,C 90.000,E1 266.216} C_DIS
LIN {X 0.015,Y -550.591,Z 584.271,A 0.000,B 0.000,C 90.000,E1 264.837} C_DIS
LIN {X -0.143,Y -549.772,Z 584.264,A 0.000,B 0.000,C 90.000,E1 263.451} C_DIS
LIN {X 0.029,Y -549.185,Z 584.259,A 0.000,B 0.000,C 90.000,E1 262.591} C_DIS
LIN {X -0.184,Y -548.152,Z 584.253,A 0.000,B 0.000,C 90.000,E1 261.489} C_DIS
LIN {X 0.232,Y -546.769,Z 584.245,A 0.000,B 0.000,C 90.000,E1 260.038} C_DIS
LIN {X -0.163,Y -544.866,Z 584.234,A 0.000,B 0.000,C 90.000,E1 258.105} C_DIS
LIN {X -0.241,Y -543.409,Z 584.226,A 0.000,B 0.000,C 90.000,E1 256.700} C_DIS
LIN {X -0.076,Y -541.338,Z 584.215,A 0.000,B 0.000,C 90.000,E1 254.700} C_DIS
LIN {X 0.252,Y -539.535,Z 584.206,A 0.000,B 0.000,C 90.000,E1 252.960} C_DIS
LIN {X 0.281,Y -538.220,Z 584.199,A 0.000,B 0.000,C 90.000,E1 251.819} C_DIS
LIN {X -0.221,Y -536.705,Z 584.193,A 0.000,B 0.000,C 90.000,E1 250.732} C_DIS
LIN {X -0.060,Y -534.911,Z 584.187,A 0.000,B 0.000,C 90.000,E1 249.571} C_DIS
LIN {X 0.072,Y -532.937,Z 584.180,A 0.000,B 0.000,C 90.000,E1 248.411} C_DIS
LIN {X 0.175,Y -531.278,Z 584.175,A 0.000,B 0.000,C 90.000,E1 247.539} C_DIS
LIN {X 0.148,Y -528.350,Z 584.167,A 0.000,B 0.000,C 90.000,E1 246.102} C_DIS
LIN {X 0.064,Y -525.335,Z 584.159,A 0.000,B 0.000,C 90.000,E1 244.665} C_DIS
LIN {X 0.140,Y -522.160,Z 584.151,A 0.000,B 0.000,C 90.000,E1 243.204} C_DIS
LIN {X -0.070,Y -518.769,Z 584.143,A 0.000,B 0.000,C 90.000,E1 241.769} C_DIS
LIN {X 0.004,Y -515.828,Z 584.137,A 0.000,B 0.000,C 90.000,E1 240.589} C_DIS
LIN {X -0.058,Y -511.931,Z 584.128,A 0.000,B 0.000,C 90.000,E1 239.125} C_DIS
LIN {X 0.134,Y -507.267,Z 584.119,A 0.000,B 0.000,C 90.000,E1 237.327} C_DIS
LIN {X -0.139,Y -504.038,Z 584.112,A 0.000,B 0.000,C 90.000,E1 236.167} C_DIS
LIN {X -0.176,Y -500.604,Z 584.105,A 0.000,B 0.000,C 90.000,E1 234.975} C_DIS
LIN {X 0.301,Y -492.356,Z 584.089,A 0.000,B 0.000,C 90.000,E1 231.904} C_DIS
LIN {X -0.034,Y -485.920,Z 584.075,A 0.000,B 0.000,C 90.000,E1 229.504} C_DIS
LIN {X -0.232,Y -479.672,Z 584.061,A 0.000,B 0.000,C 90.000,E1 227.067} C_DIS
LIN {X 0.247,Y -474.360,Z 584.049,A 0.000,B 0.000,C 90.000,E1 224.838} C_DIS
LIN {X 0.062,Y -470.678,Z 584.041,A 0.000,B 0.000,C 90.000,E1 223.299} C_DIS
LIN {X -0.102,Y -466.372,Z 584.030,A 0.000,B 0.000,C 90.000,E1 221.434} C_DIS
LIN {X 0.082,Y -461.572,Z 584.018,A 0.000,B 0.000,C 90.000,E1 219.197} C_DIS
LIN {X 0.111,Y -457.601,Z 584.007,A 0.000,B 0.000,C 90.000,E1 217.282} C_DIS
LIN {X -0.064,Y -452.320,Z 583.993,A 0.000,B 0.000,C 90.000,E1 214.739} C_DIS
LIN {X -0.059,Y -448.553,Z 583.982,A 0.000,B 0.000,C 90.000,E1 212.801} C_DIS
LIN {X -0.113,Y -443.858,Z 583.968,A 0.000,B 0.000,C 90.000,E1 210.207} C_DIS
LIN {X -0.009,Y -440.329,Z 583.957,A 0.000,B 0.000,C 90.000,E1 208.231} C_DIS
LIN {X -0.233,Y -437.440,Z 583.948,A 0.000,B 0.000,C 90.000,E1 206.616} C_DIS
LIN {X -0.125,Y -434.588,Z 583.939,A 0.000,B 0.000,C 90.000,E1 204.951} C_DIS
LIN {X 0.132,Y -431.822,Z 583.929,A 0.000,B 0.000,C 90.000,E1 203.259} C_DIS
LIN {X 0.179,Y -428.121,Z 583.916,A 0.000,B 0.000,C 90.000,E1 200.918} C_DIS
LIN {X -0.024,Y -424.621,Z 583.903,A 0.000,B 0.000,C 90.000,E1 198.598} C_DIS
LIN {X 0.043,Y -420.484,Z 583.886,A 0.000,B 0.000,C 90.000,E1 195.552} C_DIS
LIN {X 0.090,Y -418.732,Z 583.879,A 0.000,B 0.000,C 90.000,E1 194.189} C_DIS
LIN {X 0.105,Y -416.843,Z 583.871,A 0.000,B 0.000,C 90.000,E1 192.827} C_DIS
LIN {X 0.041,Y -414.338,Z 583.862,A 0.000,B 0.000,C 90.000,E1 191.130} C_DIS
LIN {X -0.005,Y -410.445,Z 583.845,A 0.000,B 0.000,C 90.000,E1 188.049} C_DIS
LIN {X 0.051,Y -408.832,Z 583.837,A 0.000,B 0.000,C 90.000,E1 186.663} C_DIS
LIN {X 0.058,Y -406.370,Z 583.826,A 0.000,B 0.000,C 90.000,E1 184.588} C_DIS
LIN {X 0.081,Y -401.767,Z 583.799,A 0.000,B 0.000,C 90.000,E1 179.714} C_DIS
LIN {X 0.148,Y -399.979,Z 583.783,A 0.000,B 0.000,C 90.000,E1 176.906} C_DIS
LIN {X 0.199,Y -398.683,Z 583.765,A 0.000,B 0.000,C 90.000,E1 173.742} C_DIS
LIN {X -0.052,Y -398.188,Z 583.752,A 0.000,B 0.000,C 90.000,E1 171.319} C_DIS
LIN {X -0.130,Y -398.029,Z 583.738,A 0.000,B 0.000,C 90.000,E1 168.870} C_DIS
LIN {X -0.085,Y -398.438,Z 583.721,A 0.000,B 0.000,C 90.000,E1 165.700} C_DIS
LIN {X 0.225,Y -399.056,Z 583.707,A 0.000,B 0.000,C 90.000,E1 163.196} C_DIS
LIN {X -0.089,Y -399.896,Z 583.693,A 0.000,B 0.000,C 90.000,E1 160.786} C_DIS
LIN {X 0.030,Y -400.801,Z 583.682,A 0.000,B 0.000,C 90.000,E1 158.666} C_DIS
LIN {X -0.050,Y -401.941,Z 583.668,A 0.000,B 0.000,C 90.000,E1 156.230} C_DIS
LIN {X 0.113,Y -402.828,Z 583.658,A 0.000,B 0.000,C 90.000,E1 154.460} C_DIS
LIN {X 0.181,Y -403.876,Z 583.647,A 0.000,B 0.000,C 90.000,E1 152.359} C_DIS
LIN {X -0.064,Y -404.540,Z 583.639,A 0.000,B 0.000,C 90.000,E1 151.001} C_DIS
LIN {X 0.006,Y -405.270,Z 583.629,A 0.000,B 0.000,C 90.000,E1 149.253} C_DIS
LIN {X -0.022,Y -405.754,Z 583.622,A 0.000,B 0.000,C 90.000,E1 147.867} C_DIS
LIN {X -0.045,Y -406.202,Z 583.612,A 0.000,B 0.000,C 90.000,E1 146.135} C_DIS
LIN {X -0.055,Y -406.606,Z 583.602,A 0.000,B 0.000,C 90.000,E1 144.402} C_DIS
LIN {X 0.173,Y -406.968,Z 583.593,A 0.000,B 0.000,C 90.000,E1 142.637} C_DIS
LIN {X -0.101,Y -407.382,Z 583.581,A 0.000,B 0.000,C 90.000,E1 140.598} C_DIS
LIN {X 0.152,Y -407.779,Z 583.570,A 0.000,B 0.000,C 90.000,E1 138.485} C_DIS
LIN {X -0.179,Y -407.965,Z 583.562,A 0.000,B 0.000,C 90.000,E1 137.148} C_DIS
LIN {X 0.053,Y -408.180,Z 583.550,A 0.000,B 0.000,C 90.000,E1 135.040} C_DIS
LIN {X 0.136,Y -408.505,Z 583.537,A 0.000,B 0.000,C 90.000,E1 132.609} C_DIS
LIN {X -0.038,Y -408.613,Z 583.527,A 0.000,B 0.000,C 90.000,E1 130.906} C_DIS
LIN {X 0.103,Y -408.601,Z 583.522,A 0.000,B 0.000,C 90.000,E1 129.850} C_DIS
LIN {X 0.094,Y -408.477,Z 583.513,A 0.000,B 0.000,C 90.000,E1 128.382} C_DIS
LIN {X -0.145,Y -415.225,Z 583.500,A 0.000,B 0.000,C 90.000,E1 126.091} C_DIS
LIN {X -0.034,Y -416.892,Z 583.497,A 0.000,B 0.000,C 90.000,E1 125.391} C_DIS
LIN {X -0.106,Y -426.614,Z 583.476,A 0.000,B 0.000,C 90.000,E1 121.671} C_DIS
LIN {X -0.143,Y -430.682,Z 583.468,A 0.000,B 0.000,C 90.000,E1 120.335} C_DIS
LIN {X -0.104,Y -431.272,Z 583.467,A 0.000,B 0.000,C 90.000,E1 120.079} C_DIS
LIN {X 0.073,Y -431.300,Z 583.467,A 0.000,B 0.000,C 90.000,E1 120.050} C_DIS
LIN {X -0.235,Y -443.388,Z 583.464,A 0.000,B 0.000,C 90.000,E1 119.539} C_DIS
LIN {X 0.048,Y -453.703,Z 583.461,A 0.000,B 0.000,C 90.000,E1 119.027} C_DIS
LIN {X 0.098,Y -469.097,Z 583.457,A 0.000,B 0.000,C 90.000,E1 118.281} C_DIS
LIN {X 0.178,Y -479.214,Z 583.454,A 0.000,B 0.000,C 90.000,E1 117.769} C_DIS
LIN {X 0.174,Y -487.441,Z 583.452,A 0.000,B 0.000,C 90.000,E1 117.334} C_DIS
LIN {X 0.028,Y -497.268,Z 583.449,A 0.000,B 0.000,C 90.000,E1 116.796} C_DIS
LIN {X 0.075,Y -505.371,Z 583.446,A 0.000,B 0.000,C 90.000,E1 116.309} C_DIS
LIN {X 0.010,Y -514.904,Z 583.443,A 0.000,B 0.000,C 90.000,E1 115.720} C_DIS
LIN {X -0.183,Y -525.379,Z 583.439,A 0.000,B 0.000,C 90.000,E1 115.027} C_DIS
LIN {X 0.184,Y -532.722,Z 583.436,A 0.000,B 0.000,C 90.000,E1 114.463} C_DIS
LIN {X 0.090,Y -538.593,Z 583.434,A 0.000,B 0.000,C 90.000,E1 114.027} C_DIS
LIN {X 0.045,Y -544.326,Z 583.431,A 0.000,B 0.000,C 90.000,E1 113.567} C_DIS
LIN {X 0.073,Y -547.137,Z 583.430,A 0.000,B 0.000,C 90.000,E1 113.334} C_DIS
LIN {X 0.296,Y -552.560,Z 583.427,A 0.000,B 0.000,C 90.000,E1 112.823} C_DIS
LIN {X 0.015,Y -557.846,Z 583.424,A 0.000,B 0.000,C 90.000,E1 112.333} C_DIS
LIN {X 0.318,Y -561.405,Z 583.422,A 0.000,B 0.000,C 90.000,E1 111.897} C_DIS
LIN {X 0.238,Y -562.668,Z 583.421,A 0.000,B 0.000,C 90.000,E1 111.770} C_DIS
LIN {X 0.075,Y -567.957,Z 583.417,A 0.000,B 0.000,C 90.000,E1 111.099} C_DIS
LIN {X -0.066,Y -572.585,Z 583.414,A 0.000,B 0.000,C 90.000,E1 110.429} C_DIS
LIN {X -0.255,Y -577.306,Z 583.409,A 0.000,B 0.000,C 90.000,E1 109.631} C_DIS
LIN {X 0.148,Y -581.641,Z 583.404,A 0.000,B 0.000,C 90.000,E1 108.779} C_DIS
LIN {X -0.218,Y -586.206,Z 583.399,A 0.000,B 0.000,C 90.000,E1 107.873} C_DIS
LIN {X -0.141,Y -588.585,Z 583.396,A 0.000,B 0.000,C 90.000,E1 107.330} C_DIS
LIN {X -0.109,Y -592.988,Z 583.390,A 0.000,B 0.000,C 90.000,E1 106.260} C_DIS
LIN {X 0.012,Y -595.163,Z 583.387,A 0.000,B 0.000,C 90.000,E1 105.717} C_DIS
LIN {X -0.308,Y -598.117,Z 583.383,A 0.000,B 0.000,C 90.000,E1 104.954} C_DIS
LIN {X 0.158,Y -602.735,Z 583.376,A 0.000,B 0.000,C 90.000,E1 103.592} C_DIS
LIN {X -0.288,Y -608.244,Z 583.367,A 0.000,B 0.000,C 90.000,E1 102.063} C_DIS
LIN {X 0.214,Y -612.864,Z 583.360,A 0.000,B 0.000,C 90.000,E1 100.715} C_DIS
LIN {X 0.319,Y -616.475,Z 583.354,A 0.000,B 0.000,C 90.000,E1 99.670} C_DIS
LIN {X -0.137,Y -619.954,Z 583.348,A 0.000,B 0.000,C 90.000,E1 98.681} C_DIS
LIN {X -0.256,Y -624.108,Z 583.341,A 0.000,B 0.000,C 90.000,E1 97.409} C_DIS
LIN {X -0.083,Y -627.336,Z 583.335,A 0.000,B 0.000,C 90.000,E1 96.372} C_DIS
LIN {X 0.134,Y -630.213,Z 583.330,A 0.000,B 0.000,C 90.000,E1 95.334} C_DIS
LIN {X -0.021,Y -632.176,Z 583.326,A 0.000,B 0.000,C 90.000,E1 94.588} C_DIS
LIN {X 0.212,Y -634.413,Z 583.320,A 0.000,B 0.000,C 90.000,E1 93.555} C_DIS
LIN {X 0.222,Y -636.755,Z 583.313,A 0.000,B 0.000,C 90.000,E1 92.293} C_DIS
LIN {X -0.260,Y -637.604,Z 583.310,A 0.000,B 0.000,C 90.000,E1 91.833} C_DIS
LIN {X 0.022,Y -638.871,Z 583.305,A 0.000,B 0.000,C 90.000,E1 90.802} C_DIS
LIN {X -0.071,Y -639.611,Z 583.300,A 0.000,B 0.000,C 90.000,E1 90.057} C_DIS
LIN {X -0.155,Y -640.099,Z 583.296,A 0.000,B 0.000,C 90.000,E1 89.312} C_DIS
LIN {X -0.238,Y -640.366,Z 583.292,A 0.000,B 0.000,C 90.000,E1 88.568} C_DIS
LIN {X 0.100,Y -640.234,Z 583.286,A 0.000,B 0.000,C 90.000,E1 87.535} C_DIS
LIN {X 0.046,Y -639.942,Z 583.282,A 0.000,B 0.000,C 90.000,E1 86.788} C_DIS
LIN {X -0.253,Y -639.224,Z 583.277,A 0.000,B 0.000,C 90.000,E1 85.812} C_DIS
LIN {X 0.323,Y -638.509,Z 583.272,A 0.000,B 0.000,C 90.000,E1 85.008} C_DIS
LIN {X -0.202,Y -636.929,Z 583.266,A 0.000,B 0.000,C 90.000,E1 83.799} C_DIS
LIN {X -0.027,Y -636.228,Z 583.263,A 0.000,B 0.000,C 90.000,E1 83.280} C_DIS
LIN {X 0.144,Y -635.358,Z 583.260,A 0.000,B 0.000,C 90.000,E1 82.761} C_DIS
LIN {X 0.265,Y -632.794,Z 583.253,A 0.000,B 0.000,C 90.000,E1 81.489} C_DIS
LIN {X -0.287,Y -629.806,Z 583.246,A 0.000,B 0.000,C 90.000,E1 80.274} C_DIS
LIN {X 0.155,Y -627.212,Z 583.240,A 0.000,B 0.000,C 90.000,E1 79.218} C_DIS
LIN {X 0.233,Y -623.636,Z 583.233,A 0.000,B 0.000,C 90.000,E1 77.937} C_DIS
LIN {X -0.011,Y -620.473,Z 583.227,A 0.000,B 0.000,C 90.000,E1 76.937} C_DIS
LIN {X -0.294,Y -617.049,Z 583.222,A 0.000,B 0.000,C 90.000,E1 75.936} C_DIS
LIN {X 0.203,Y -614.293,Z 583.217,A 0.000,B 0.000,C 90.000,E1 75.117} C_DIS
LIN {X 0.234,Y -611.332,Z 583.213,A 0.000,B 0.000,C 90.000,E1 74.338} C_DIS
LIN {X -0.059,Y -606.267,Z 583.207,A 0.000,B 0.000,C 90.000,E1 73.196} C_DIS
LIN {X -0.102,Y -602.599,Z 583.202,A 0.000,B 0.000,C 90.000,E1 72.417} C_DIS
LIN {X -0.186,Y -598.625,Z 583.198,A 0.000,B 0.000,C 90.000,E1 71.638} C_DIS
LIN {X -0.316,Y -594.335,Z 583.194,A 0.000,B 0.000,C 90.000,E1 70.859} C_DIS
LIN {X -0.295,Y -589.665,Z 583.189,A 0.000,B 0.000,C 90.000,E1 70.061} C_DIS
LIN {X -0.253,Y -585.315,Z 583.185,A 0.000,B 0.000,C 90.000,E1 69.390} C_DIS
LIN {X -0.182,Y -580.540,Z 583.182,A 0.000,B 0.000,C 90.000,E1 68.720} C_DIS
LIN {X 0.137,Y -576.455,Z 583.179,A 0.000,B 0.000,C 90.000,E1 68.156} C_DIS
LIN {X 0.137,Y -571.902,Z 583.176,A 0.000,B 0.000,C 90.000,E1 67.614} C_DIS
LIN {X 0.128,Y -566.058,Z 583.172,A 0.000,B 0.000,C 90.000,E1 66.975} C_DIS
LIN {X 0.150,Y -561.235,Z 583.169,A 0.000,B 0.000,C 90.000,E1 66.485} C_DIS
LIN {X -0.292,Y -556.006,Z 583.167,A 0.000,B 0.000,C 90.000,E1 66.049} C_DIS
LIN {X 0.116,Y -550.351,Z 583.164,A 0.000,B 0.000,C 90.000,E1 65.537} C_DIS
LIN {X -0.298,Y -545.688,Z 583.162,A 0.000,B 0.000,C 90.000,E1 65.229} C_DIS
LIN {X -0.050,Y -539.390,Z 583.160,A 0.000,B 0.000,C 90.000,E1 64.793} C_DIS
LIN {X -0.262,Y -534.721,Z 583.158,A 0.000,B 0.000,C 90.000,E1 64.537} C_DIS
LIN {X -0.041,Y -527.975,Z 583.156,A 0.000,B 0.000,C 90.000,E1 64.152} C_DIS
LIN {X 0.144,Y -519.379,Z 583.154,A 0.000,B 0.000,C 90.000,E1 63.717} C_DIS
LIN {X 0.142,Y -510.634,Z 583.152,A 0.000,B 0.000,C 90.000,E1 63.332} C_DIS
LIN {X 0.000,Y -503.618,Z 583.150,A 0.000,B 0.000,C 90.000,E1 63.050} C_DIS
LIN {X -0.052,Y -489.866,Z 583.147,A 0.000,B 0.000,C 90.000,E1 62.487} C_DIS
LIN {X 0.141,Y -466.212,Z 583.141,A 0.000,B 0.000,C 90.000,E1 61.435} C_DIS
LIN {X 0.161,Y -452.904,Z 583.138,A 0.000,B 0.000,C 90.000,E1 60.795} C_DIS
LIN {X 0.119,Y -452.799,Z 583.138,A 0.000,B 0.000,C 90.000,E1 60.795} C_DIS
LIN {X 0.079,Y -443.806,Z 583.114,A 0.000,B 0.000,C 90.000,E1 56.421} C_DIS
LIN {X -0.187,Y -434.912,Z 583.092,A 0.000,B 0.000,C 90.000,E1 52.637} C_DIS
LIN {X -0.107,Y -436.921,Z 583.081,A 0.000,B 0.000,C 90.000,E1 50.517} C_DIS
LIN {X -0.038,Y -438.817,Z 583.070,A 0.000,B 0.000,C 90.000,E1 48.528} C_DIS
LIN {X 0.077,Y -440.748,Z 583.059,A 0.000,B 0.000,C 90.000,E1 46.539} C_DIS
LIN {X -0.050,Y -442.008,Z 583.051,A 0.000,B 0.000,C 90.000,E1 45.243} C_DIS
LIN {X -0.129,Y -442.855,Z 583.046,A 0.000,B 0.000,C 90.000,E1 44.271} C_DIS
LIN {X 0.097,Y -443.764,Z 583.039,A 0.000,B 0.000,C 90.000,E1 42.933} C_DIS
LIN {X 0.040,Y -444.539,Z 583.031,A 0.000,B 0.000,C 90.000,E1 41.634} C_DIS
LIN {X -0.026,Y -445.276,Z 583.022,A 0.000,B 0.000,C 90.000,E1 40.011} C_DIS
LIN {X -0.045,Y -445.669,Z 583.017,A 0.000,B 0.000,C 90.000,E1 39.036} C_DIS
LIN {X -0.019,Y -446.044,Z 583.010,A 0.000,B 0.000,C 90.000,E1 37.729} C_DIS
LIN {X 0.011,Y -446.243,Z 583.002,A 0.000,B 0.000,C 90.000,E1 36.423} C_DIS
LIN {X 0.140,Y -446.304,Z 582.995,A 0.000,B 0.000,C 90.000,E1 35.105} C_DIS
LIN {X -0.094,Y -446.193,Z 582.988,A 0.000,B 0.000,C 90.000,E1 33.833} C_DIS
LIN {X -0.011,Y -446.065,Z 582.975,A 0.000,B 0.000,C 90.000,E1 31.544} C_DIS
LIN {X -0.088,Y -445.924,Z 582.961,A 0.000,B 0.000,C 90.000,E1 28.949} C_DIS
LIN {X -0.132,Y -445.874,Z 582.950,A 0.000,B 0.000,C 90.000,E1 27.001} C_DIS
LIN {X -0.069,Y -445.820,Z 582.935,A 0.000,B 0.000,C 90.000,E1 24.387} C_DIS
LIN {X -0.021,Y -445.961,Z 582.928,A 0.000,B 0.000,C 90.000,E1 23.078} C_DIS
LIN {X 0.044,Y -446.155,Z 582.916,A 0.000,B 0.000,C 90.000,E1 20.791} C_DIS
LIN {X -0.065,Y -446.439,Z 582.905,A 0.000,B 0.000,C 90.000,E1 18.852} C_DIS
LIN {X -0.010,Y -446.873,Z 582.892,A 0.000,B 0.000,C 90.000,E1 16.567} C_DIS
LIN {X -0.074,Y -447.604,Z 582.879,A 0.000,B 0.000,C 90.000,E1 14.300} C_DIS
LIN {X -0.163,Y -448.722,Z 582.865,A 0.000,B 0.000,C 90.000,E1 11.715} C_DIS
LIN {X -0.069,Y -449.974,Z 582.852,A 0.000,B 0.000,C 90.000,E1 9.434} C_DIS
LIN {X -0.160,Y -451.475,Z 582.840,A 0.000,B 0.000,C 90.000,E1 7.182} C_DIS
LIN {X 0.112,Y -453.846,Z 582.824,A 0.000,B 0.000,C 90.000,E1 4.245} C_DIS
LIN {X 0.020,Y -455.996,Z 582.811,A 0.000,B 0.000,C 90.000,E1 2.007} C_DIS
LIN {X -0.092,Y -458.821,Z 582.797,A 0.000,B 0.000,C 90.000,E1 359.484} C_DIS
LIN {X 0.134,Y -462.156,Z 582.783,A 0.000,B 0.000,C 90.000,E1 356.906} C_DIS
LIN {X -0.162,Y -464.457,Z 582.774,A 0.000,B 0.000,C 90.000,E1 355.355} C_DIS
LIN {X 0.104,Y -467.729,Z 582.762,A 0.000,B 0.000,C 90.000,E1 353.109} C_DIS
LIN {X 0.204,Y -469.698,Z 582.755,A 0.000,B 0.000,C 90.000,E1 351.837} C_DIS
LIN {X 0.156,Y -472.135,Z 582.746,A 0.000,B 0.000,C 90.000,E1 350.274} C_DIS
LIN {X -0.101,Y -475.517,Z 582.734,A 0.000,B 0.000,C 90.000,E1 348.117} C_DIS
LIN {X -0.218,Y -479.651,Z 582.720,A 0.000,B 0.000,C 90.000,E1 345.644} C_DIS
LIN {X 0.044,Y -484.097,Z 582.706,A 0.000,B 0.000,C 90.000,E1 343.142} C_DIS
LIN {X -0.241,Y -486.403,Z 582.700,A 0.000,B 0.000,C 90.000,E1 341.945} C_DIS
LIN {X 0.142,Y -489.380,Z 582.691,A 0.000,B 0.000,C 90.000,E1 340.369} C_DIS
LIN {X 0.119,Y -492.324,Z 582.683,A 0.000,B 0.000,C 90.000,E1 338.847} C_DIS
LIN {X -0.131,Y -495.114,Z 582.674,A 0.000,B 0.000,C 90.000,E1 337.358} C_DIS
LIN {X 0.270,Y -497.279,Z 582.667,A 0.000,B 0.000,C 90.000,E1 336.102} C_DIS
LIN {X 0.105,Y -499.810,Z 582.659,A 0.000,B 0.000,C 90.000,E1 334.613} C_DIS
LIN {X 0.023,Y -502.718,Z 582.649,A 0.000,B 0.000,C 90.000,E1 332.820} C_DIS
LIN {X 0.109,Y -505.974,Z 582.637,A 0.000,B 0.000,C 90.000,E1 330.717} C_DIS
LIN {X -0.151,Y -509.314,Z 582.626,A 0.000,B 0.000,C 90.000,E1 328.663} C_DIS
LIN {X 0.297,Y -512.242,Z 582.616,A 0.000,B 0.000,C 90.000,E1 326.834} C_DIS
LIN {X -0.117,Y -515.876,Z 582.604,A 0.000,B 0.000,C 90.000,E1 324.815} C_DIS
LIN {X -0.023,Y -518.522,Z 582.596,A 0.000,B 0.000,C 90.000,E1 323.336} C_DIS
LIN {X -0.080,Y -522.334,Z 582.585,A 0.000,B 0.000,C 90.000,E1 321.295} C_DIS
LIN {X -0.008,Y -525.727,Z 582.575,A 0.000,B 0.000,C 90.000,E1 319.542} C_DIS
LIN {X -0.214,Y -528.238,Z 582.569,A 0.000,B 0.000,C 90.000,E1 318.405} C_DIS
LIN {X -0.059,Y -532.090,Z 582.561,A 0.000,B 0.000,C 90.000,E1 316.944} C_DIS
LIN {X -0.138,Y -533.886,Z 582.558,A 0.000,B 0.000,C 90.000,E1 316.377} C_DIS
LIN {X -0.338,Y -535.744,Z 582.555,A 0.000,B 0.000,C 90.000,E1 315.972} C_DIS
LIN {X 0.004,Y -537.537,Z 582.554,A 0.000,B 0.000,C 90.000,E1 315.648} C_DIS
LIN {X 0.185,Y -538.310,Z 582.553,A 0.000,B 0.000,C 90.000,E1 315.486} C_DIS
LIN {X 0.028,Y -540.671,Z 582.551,A 0.000,B 0.000,C 90.000,E1 315.202} C_DIS
LIN {X 0.016,Y -542.755,Z 582.550,A 0.000,B 0.000,C 90.000,E1 314.919} C_DIS
LIN {X -0.287,Y -546.894,Z 582.547,A 0.000,B 0.000,C 90.000,E1 314.514} C_DIS
LIN {X -0.361,Y -551.548,Z 582.545,A 0.000,B 0.000,C 90.000,E1 314.109} C_DIS
LIN {X 0.123,Y -559.661,Z 582.541,A 0.000,B 0.000,C 90.000,E1 313.419} C_DIS
LIN {X 0.081,Y -573.090,Z 582.536,A 0.000,B 0.000,C 90.000,E1 312.447} C_DIS
LIN {X -0.165,Y -586.302,Z 582.531,A 0.000,B 0.000,C 90.000,E1 311.515} C_DIS
LIN {X -0.278,Y -590.603,Z 582.529,A 0.000,B 0.000,C 90.000,E1 311.229} C_DIS
LIN {X -0.037,Y -596.294,Z 582.527,A 0.000,B 0.000,C 90.000,E1 310.782} C_DIS
LIN {X -0.107,Y -600.465,Z 582.525,A 0.000,B 0.000,C 90.000,E1 310.458} C_DIS
LIN {X 0.136,Y -604.595,Z 582.523,A 0.000,B 0.000,C 90.000,E1 310.092} C_DIS
LIN {X 0.275,Y -611.040,Z 582.520,A 0.000,B 0.000,C 90.000,E1 309.483} C_DIS
LIN {X -0.233,Y -616.067,Z 582.517,A 0.000,B 0.000,C 90.000,E1 309.036} C_DIS
LIN {X -0.071,Y -620.906,Z 582.514,A 0.000,B 0.000,C 90.000,E1 308.508} C_DIS
LIN {X 0.062,Y -626.696,Z 582.510,A 0.000,B 0.000,C 90.000,E1 307.855} C_DIS
LIN {X -0.047,Y -633.929,Z 582.506,A 0.000,B 0.000,C 90.000,E1 306.996} C_DIS
LIN {X -0.182,Y -638.906,Z 582.502,A 0.000,B 0.000,C 90.000,E1 306.377} C_DIS
LIN {X 0.142,Y -645.331,Z 582.497,A 0.000,B 0.000,C 90.000,E1 305.471} C_DIS
LIN {X 0.085,Y -648.820,Z 582.494,A 0.000,B 0.000,C 90.000,E1 304.978} C_DIS
LIN {X -0.048,Y -653.402,Z 582.490,A 0.000,B 0.000,C 90.000,E1 304.246} C_DIS
LIN {X 0.077,Y -655.587,Z 582.488,A 0.000,B 0.000,C 90.000,E1 303.865} C_DIS
LIN {X 0.133,Y -658.787,Z 582.485,A 0.000,B 0.000,C 90.000,E1 303.245} C_DIS
LIN {X -0.289,Y -662.244,Z 582.481,A 0.000,B 0.000,C 90.000,E1 302.546} C_DIS
LIN {X -0.125,Y -665.471,Z 582.477,A 0.000,B 0.000,C 90.000,E1 301.799} C_DIS
LIN {X 0.219,Y -669.587,Z 582.471,A 0.000,B 0.000,C 90.000,E1 300.797} C_DIS
LIN {X 0.116,Y -672.597,Z 582.467,A 0.000,B 0.000,C 90.000,E1 300.079} C_DIS
LIN {X -0.034,Y -676.263,Z 582.462,A 0.000,B 0.000,C 90.000,E1 299.127} C_DIS
LIN {X -0.075,Y -678.791,Z 582.458,A 0.000,B 0.000,C 90.000,E1 298.409} C_DIS
LIN {X -0.002,Y -682.655,Z 582.451,A 0.000,B 0.000,C 90.000,E1 297.206} C_DIS
LIN {X -0.192,Y -684.066,Z 582.449,A 0.000,B 0.000,C 90.000,E1 296.744} C_DIS
LIN {X 0.021,Y -684.674,Z 582.447,A 0.000,B 0.000,C 90.000,E1 296.488} C_DIS
LIN {X -0.163,Y -685.389,Z 582.445,A 0.000,B 0.000,C 90.000,E1 296.027} C_DIS
LIN {X 0.054,Y -685.524,Z 582.443,A 0.000,B 0.000,C 90.000,E1 295.771} C_DIS
LIN {X 0.196,Y -684.656,Z 582.441,A 0.000,B 0.000,C 90.000,E1 295.283} C_DIS
LIN {X -0.205,Y -683.871,Z 582.439,A 0.000,B 0.000,C 90.000,E1 295.079} C_DIS
LIN {X -0.097,Y -683.270,Z 582.439,A 0.000,B 0.000,C 90.000,E1 294.951} C_DIS
LIN {X 0.010,Y -682.300,Z 582.438,A 0.000,B 0.000,C 90.000,E1 294.823} C_DIS
LIN {X -0.065,Y -679.984,Z 582.437,A 0.000,B 0.000,C 90.000,E1 294.591} C_DIS
LIN {X 0.137,Y -677.696,Z 582.435,A 0.000,B 0.000,C 90.000,E1 294.335} C_DIS
LIN {X 0.250,Y -675.804,Z 582.435,A 0.000,B 0.000,C 90.000,E1 294.207} C_DIS
LIN {X 0.072,Y -669.845,Z 582.433,A 0.000,B 0.000,C 90.000,E1 293.951} C_DIS
LIN {X -0.139,Y -668.244,Z 582.433,A 0.000,B 0.000,C 90.000,E1 293.898} C_DIS
LIN {X 0.143,Y -662.223,Z 582.432,A 0.000,B 0.000,C 90.000,E1 293.695} C_DIS
LIN {X 0.156,Y -660.164,Z 582.431,A 0.000,B 0.000,C 90.000,E1 293.643} C_DIS
LIN {X 0.081,Y -650.080,Z 582.430,A 0.000,B 0.000,C 90.000,E1 293.462} C_DIS
LIN {X -0.039,Y -633.421,Z 582.429,A 0.000,B 0.000,C 90.000,E1 293.131} C_DIS
LIN {X 0.316,Y -620.148,Z 582.427,A 0.000,B 0.000,C 90.000,E1 292.770} C_DIS
LIN {X 0.063,Y -610.169,Z 582.425,A 0.000,B 0.000,C 90.000,E1 292.514} C_DIS
LIN {X 0.044,Y -579.182,Z 582.420,A 0.000,B 0.000,C 90.000,E1 291.535} C_DIS
LIN {X 0.322,Y -572.152,Z 582.418,A 0.000,B 0.000,C 90.000,E1 291.280} C_DIS
LIN {X -0.068,Y -566.885,Z 582.417,A 0.000,B 0.000,C 90.000,E1 291.099} C_DIS
LIN {X -0.215,Y -564.562,Z 582.416,A 0.000,B 0.000,C 90.000,E1 290.972} C_DIS
LIN {X 0.188,Y -562.431,Z 582.416,A 0.000,B 0.000,C 90.000,E1 290.791} C_DIS
LIN {X 0.156,Y -562.382,Z 582.416,A 0.000,B 0.000,C 90.000,E1 290.791} C_DIS
LIN {X 0.090,Y -561.701,Z 582.415,A 0.000,B 0.000,C 90.000,E1 290.663} C_DIS
LIN {X -0.166,Y -561.329,Z 582.414,A 0.000,B 0.000,C 90.000,E1 290.482} C_DIS
LIN {X 0.147,Y -561.000,Z 582.412,A 0.000,B 0.000,C 90.000,E1 290.174} C_DIS
LIN {X -0.144,Y -561.171,Z 582.405,A 0.000,B 0.000,C 90.000,E1 288.833} C_DIS
LIN {X -0.202,Y -560.813,Z 582.397,A 0.000,B 0.000,C 90.000,E1 287.457} C_DIS
LIN {X 0.136,Y -560.414,Z 582.391,A 0.000,B 0.000,C 90.000,E1 286.315} C_DIS
LIN {X 0.171,Y -560.085,Z 582.386,A 0.000,B 0.000,C 90.000,E1 285.481} C_DIS
LIN {X 0.087,Y -559.170,Z 582.377,A 0.000,B 0.000,C 90.000,E1 283.828} C_DIS
LIN {X 0.119,Y -558.535,Z 582.371,A 0.000,B 0.000,C 90.000,E1 282.715} C_DIS
LIN {X -0.114,Y -557.614,Z 582.362,A 0.000,B 0.000,C 90.000,E1 281.074} C_DIS
LIN {X 0.166,Y -556.633,Z 582.352,A 0.000,B 0.000,C 90.000,E1 279.378} C_DIS
LIN {X -0.188,Y -555.686,Z 582.341,A 0.000,B 0.000,C 90.000,E1 277.466} C_DIS
LIN {X -0.144,Y -554.801,Z 582.331,A 0.000,B 0.000,C 90.000,E1 275.511} C_DIS
LIN {X -0.042,Y -554.087,Z 582.318,A 0.000,B 0.000,C 90.000,E1 273.269} C_DIS
LIN {X -0.138,Y -553.640,Z 582.309,A 0.000,B 0.000,C 90.000,E1 271.604} C_DIS
LIN {X 0.272,Y -553.075,Z 582.300,A 0.000,B 0.000,C 90.000,E1 269.885} C_DIS
LIN {X 0.114,Y -552.387,Z 582.290,A 0.000,B 0.000,C 90.000,E1 268.224} C_DIS
LIN {X -0.021,Y -551.710,Z 582.281,A 0.000,B 0.000,C 90.000,E1 266.560} C_DIS
LIN {X -0.212,Y -551.033,Z 582.273,A 0.000,B 0.000,C 90.000,E1 265.179} C_DIS
LIN {X 0.130,Y -550.238,Z 582.265,A 0.000,B 0.000,C 90.000,E1 263.742} C_DIS
LIN {X -0.138,Y -549.495,Z 582.259,A 0.000,B 0.000,C 90.000,E1 262.648} C_DIS
LIN {X 0.199,Y -548.463,Z 582.253,A 0.000,B 0.000,C 90.000,E1 261.489} C_DIS
LIN {X -0.021,Y -547.380,Z 582.247,A 0.000,B 0.000,C 90.000,E1 260.387} C_DIS
LIN {X 0.119,Y -545.179,Z 582.234,A 0.000,B 0.000,C 90.000,E1 258.117} C_DIS
LIN {X 0.243,Y -543.418,Z 582.225,A 0.000,B 0.000,C 90.000,E1 256.408} C_DIS
LIN {X -0.194,Y -541.621,Z 582.215,A 0.000,B 0.000,C 90.000,E1 254.755} C_DIS
LIN {X -0.073,Y -540.139,Z 582.207,A 0.000,B 0.000,C 90.000,E1 253.323} C_DIS
LIN {X -0.037,Y -538.824,Z 582.201,A 0.000,B 0.000,C 90.000,E1 252.181} C_DIS
LIN {X 0.193,Y -536.908,Z 582.193,A 0.000,B 0.000,C 90.000,E1 250.732} C_DIS
LIN {X -0.146,Y -535.124,Z 582.187,A 0.000,B 0.000,C 90.000,E1 249.625} C_DIS
LIN {X 0.196,Y -532.653,Z 582.179,A 0.000,B 0.000,C 90.000,E1 248.156} C_DIS
LIN {X 0.172,Y -529.154,Z 582.169,A 0.000,B 0.000,C 90.000,E1 246.433} C_DIS
LIN {X 0.317,Y -526.144,Z 582.161,A 0.000,B 0.000,C 90.000,E1 244.973} C_DIS
LIN {X -0.057,Y -522.971,Z 582.153,A 0.000,B 0.000,C 90.000,E1 243.563} C_DIS
LIN {X -0.023,Y -519.627,Z 582.145,A 0.000,B 0.000,C 90.000,E1 242.103} C_DIS
LIN {X -0.059,Y -517.478,Z 582.140,A 0.000,B 0.000,C 90.000,E1 241.229} C_DIS
LIN {X 0.002,Y -514.412,Z 582.134,A 0.000,B 0.000,C 90.000,E1 240.049} C_DIS
LIN {X 0.010,Y -511.256,Z 582.127,A 0.000,B 0.000,C 90.000,E1 238.869} C_DIS
LIN {X -0.247,Y -506.562,Z 582.117,A 0.000,B 0.000,C 90.000,E1 237.120} C_DIS
LIN {X 0.170,Y -503.255,Z 582.111,A 0.000,B 0.000,C 90.000,E1 235.881} C_DIS
LIN {X 0.122,Y -499.813,Z 582.104,A 0.000,B 0.000,C 90.000,E1 234.689} C_DIS
LIN {X 0.023,Y -492.428,Z 582.089,A 0.000,B 0.000,C 90.000,E1 231.984} C_DIS
LIN {X 0.204,Y -485.193,Z 582.074,A 0.000,B 0.000,C 90.000,E1 229.218} C_DIS
LIN {X 0.176,Y -479.721,Z 582.062,A 0.000,B 0.000,C 90.000,E1 227.067} C_DIS
LIN {X -0.126,Y -475.172,Z 582.051,A 0.000,B 0.000,C 90.000,E1 225.243} C_DIS
LIN {X -0.201,Y -470.727,Z 582.041,A 0.000,B 0.000,C 90.000,E1 223.380} C_DIS
LIN {X -0.011,Y -466.421,Z 582.030,A 0.000,B 0.000,C 90.000,E1 221.472} C_DIS
LIN {X -0.171,Y -461.617,Z 582.018,A 0.000,B 0.000,C 90.000,E1 219.277} C_DIS
LIN {X -0.136,Y -457.612,Z 582.008,A 0.000,B 0.000,C 90.000,E1 217.363} C_DIS
LIN {X 0.069,Y -452.321,Z 581.993,A 0.000,B 0.000,C 90.000,E1 214.771} C_DIS
LIN {X -0.215,Y -447.928,Z 581.981,A 0.000,B 0.000,C 90.000,E1 212.546} C_DIS
LIN {X -0.114,Y -443.815,Z 581.968,A 0.000,B 0.000,C 90.000,E1 210.256} C_DIS
LIN {X -0.063,Y -440.860,Z 581.959,A 0.000,B 0.000,C 90.000,E1 208.615} C_DIS
LIN {X 0.114,Y -438.005,Z 581.950,A 0.000,B 0.000,C 90.000,E1 206.950} C_DIS
LIN {X 0.065,Y -434.567,Z 581.939,A 0.000,B 0.000,C 90.000,E1 204.975} C_DIS
LIN {X -0.066,Y -431.787,Z 581.930,A 0.000,B 0.000,C 90.000,E1 203.334} C_DIS
LIN {X 0.145,Y -428.095,Z 581.917,A 0.000,B 0.000,C 90.000,E1 200.972} C_DIS
LIN {X -0.064,Y -424.626,Z 581.904,A 0.000,B 0.000,C 90.000,E1 198.652} C_DIS
LIN {X -0.060,Y -420.927,Z 581.889,A 0.000,B 0.000,C 90.000,E1 195.953} C_DIS
LIN {X -0.015,Y -419.234,Z 581.881,A 0.000,B 0.000,C 90.000,E1 194.592} C_DIS
LIN {X 0.056,Y -416.907,Z 581.872,A 0.000,B 0.000,C 90.000,E1 192.883} C_DIS
LIN {X 0.167,Y -412.563,Z 581.855,A 0.000,B 0.000,C 90.000,E1 189.792} C_DIS
LIN {X 0.000,Y -409.720,Z 581.841,A 0.000,B 0.000,C 90.000,E1 187.409} C_DIS
LIN {X 0.024,Y -407.265,Z 581.830,A 0.000,B 0.000,C 90.000,E1 185.334} C_DIS
LIN {X -0.172,Y -403.543,Z 581.810,A 0.000,B 0.000,C 90.000,E1 181.892} C_DIS
LIN {X -0.084,Y -401.152,Z 581.793,A 0.000,B 0.000,C 90.000,E1 178.740} C_DIS
LIN {X 0.029,Y -399.688,Z 581.779,A 0.000,B 0.000,C 90.000,E1 176.274} C_DIS
LIN {X 0.098,Y -398.740,Z 581.764,A 0.000,B 0.000,C 90.000,E1 173.457} C_DIS
LIN {X -0.123,Y -398.221,Z 581.748,A 0.000,B 0.000,C 90.000,E1 170.679} C_DIS
LIN {X -0.175,Y -398.145,Z 581.736,A 0.000,B 0.000,C 90.000,E1 168.578} C_DIS
LIN {X -0.101,Y -398.548,Z 581.721,A 0.000,B 0.000,C 90.000,E1 165.755} C_DIS
LIN {X 0.103,Y -399.165,Z 581.707,A 0.000,B 0.000,C 90.000,E1 163.268} C_DIS
LIN {X -0.220,Y -400.028,Z 581.694,A 0.000,B 0.000,C 90.000,E1 160.859} C_DIS
LIN {X 0.121,Y -401.101,Z 581.680,A 0.000,B 0.000,C 90.000,E1 158.358} C_DIS
LIN {X 0.050,Y -402.251,Z 581.666,A 0.000,B 0.000,C 90.000,E1 155.921} C_DIS
LIN {X -0.147,Y -403.133,Z 581.657,A 0.000,B 0.000,C 90.000,E1 154.204} C_DIS
LIN {X 0.032,Y -404.049,Z 581.647,A 0.000,B 0.000,C 90.000,E1 152.436} C_DIS
LIN {X -0.018,Y -404.710,Z 581.639,A 0.000,B 0.000,C 90.000,E1 151.051} C_DIS
LIN {X -0.146,Y -405.468,Z 581.630,A 0.000,B 0.000,C 90.000,E1 149.331} C_DIS
LIN {X 0.042,Y -405.983,Z 581.622,A 0.000,B 0.000,C 90.000,E1 147.916} C_DIS
LIN {X 0.275,Y -406.511,Z 581.610,A 0.000,B 0.000,C 90.000,E1 145.801} C_DIS
LIN {X -0.063,Y -406.907,Z 581.601,A 0.000,B 0.000,C 90.000,E1 144.116} C_DIS
LIN {X -0.153,Y -407.239,Z 581.591,A 0.000,B 0.000,C 90.000,E1 142.396} C_DIS
LIN {X 0.011,Y -407.571,Z 581.581,A 0.000,B 0.000,C 90.000,E1 140.642} C_DIS
LIN {X 0.009,Y -407.931,Z 581.570,A 0.000,B 0.000,C 90.000,E1 138.566} C_DIS
LIN {X -0.021,Y -408.149,Z 581.562,A 0.000,B 0.000,C 90.000,E1 137.187} C_DIS
LIN {X 0.050,Y -408.344,Z 581.549,A 0.000,B 0.000,C 90.000,E1 134.757} C_DIS
LIN {X 0.157,Y -408.577,Z 581.539,A 0.000,B 0.000,C 90.000,E1 133.014} C_DIS
LIN {X -0.011,Y -408.772,Z 581.530,A 0.000,B 0.000,C 90.000,E1 131.310} C_DIS
LIN {X -0.024,Y -408.749,Z 581.522,A 0.000,B 0.000,C 90.000,E1 129.930} C_DIS
LIN {X -0.072,Y -408.544,Z 581.513,A 0.000,B 0.000,C 90.000,E1 128.382} C_DIS
LIN {X -0.025,Y -415.031,Z 581.501,A 0.000,B 0.000,C 90.000,E1 126.137} C_DIS
LIN {X -0.095,Y -415.971,Z 581.499,A 0.000,B 0.000,C 90.000,E1 125.804} C_DIS
LIN {X 0.011,Y -425.467,Z 581.478,A 0.000,B 0.000,C 90.000,E1 122.054} C_DIS
LIN {X -0.054,Y -430.491,Z 581.469,A 0.000,B 0.000,C 90.000,E1 120.384} C_DIS
LIN {X 0.065,Y -431.858,Z 581.466,A 0.000,B 0.000,C 90.000,E1 119.795} C_DIS
LIN {X 0.025,Y -431.971,Z 581.466,A 0.000,B 0.000,C 90.000,E1 119.795} C_DIS
LIN {X -0.233,Y -451.247,Z 581.461,A 0.000,B 0.000,C 90.000,E1 118.949} C_DIS
LIN {X 0.015,Y -468.351,Z 581.456,A 0.000,B 0.000,C 90.000,E1 118.103} C_DIS
LIN {X 0.185,Y -478.324,Z 581.453,A 0.000,B 0.000,C 90.000,E1 117.590} C_DIS
LIN {X 0.086,Y -484.969,Z 581.452,A 0.000,B 0.000,C 90.000,E1 117.257} C_DIS
LIN {X -0.059,Y -491.475,Z 581.450,A 0.000,B 0.000,C 90.000,E1 116.924} C_DIS
LIN {X -0.222,Y -499.429,Z 581.447,A 0.000,B 0.000,C 90.000,E1 116.488} C_DIS
LIN {X 0.126,Y -507.382,Z 581.444,A 0.000,B 0.000,C 90.000,E1 115.976} C_DIS
LIN {X -0.203,Y -515.066,Z 581.442,A 0.000,B 0.000,C 90.000,E1 115.540} C_DIS
LIN {X 0.222,Y -523.943,Z 581.439,A 0.000,B 0.000,C 90.000,E1 114.899} C_DIS
LIN {X 0.128,Y -531.491,Z 581.436,A 0.000,B 0.000,C 90.000,E1 114.387} C_DIS
LIN {X 0.091,Y -537.380,Z 581.433,A 0.000,B 0.000,C 90.000,E1 113.951} C_DIS
LIN {X -0.259,Y -541.867,Z 581.431,A 0.000,B 0.000,C 90.000,E1 113.643} C_DIS
LIN {X 0.053,Y -547.371,Z 581.429,A 0.000,B 0.000,C 90.000,E1 113.153} C_DIS
LIN {X -0.044,Y -552.445,Z 581.426,A 0.000,B 0.000,C 90.000,E1 112.717} C_DIS
LIN {X 0.303,Y -557.431,Z 581.424,A 0.000,B 0.000,C 90.000,E1 112.206} C_DIS
LIN {X -0.185,Y -562.406,Z 581.421,A 0.000,B 0.000,C 90.000,E1 111.716} C_DIS
LIN {X -0.147,Y -567.772,Z 581.417,A 0.000,B 0.000,C 90.000,E1 111.025} C_DIS
LIN {X 0.241,Y -572.495,Z 581.413,A 0.000,B 0.000,C 90.000,E1 110.301} C_DIS
LIN {X -0.227,Y -578.163,Z 581.408,A 0.000,B 0.000,C 90.000,E1 109.396} C_DIS
LIN {X 0.189,Y -582.495,Z 581.403,A 0.000,B 0.000,C 90.000,E1 108.544} C_DIS
LIN {X -0.162,Y -587.065,Z 581.398,A 0.000,B 0.000,C 90.000,E1 107.638} C_DIS
LIN {X -0.220,Y -592.309,Z 581.391,A 0.000,B 0.000,C 90.000,E1 106.441} C_DIS
LIN {X 0.166,Y -595.581,Z 581.387,A 0.000,B 0.000,C 90.000,E1 105.607} C_DIS
LIN {X 0.009,Y -598.601,Z 581.382,A 0.000,B 0.000,C 90.000,E1 104.828} C_DIS
LIN {X 0.031,Y -602.414,Z 581.377,A 0.000,B 0.000,C 90.000,E1 103.772} C_DIS
LIN {X -0.085,Y -608.896,Z 581.366,A 0.000,B 0.000,C 90.000,E1 101.951} C_DIS
LIN {X 0.186,Y -614.495,Z 581.358,A 0.000,B 0.000,C 90.000,E1 100.366} C_DIS
LIN {X 0.315,Y -618.123,Z 581.352,A 0.000,B 0.000,C 90.000,E1 99.321} C_DIS
LIN {X 0.115,Y -620.739,Z 581.348,A 0.000,B 0.000,C 90.000,E1 98.568} C_DIS
LIN {X -0.293,Y -625.762,Z 581.339,A 0.000,B 0.000,C 90.000,E1 97.068} C_DIS
LIN {X 0.202,Y -628.159,Z 581.335,A 0.000,B 0.000,C 90.000,E1 96.258} C_DIS
LIN {X -0.194,Y -631.074,Z 581.329,A 0.000,B 0.000,C 90.000,E1 95.277} C_DIS
LIN {X 0.290,Y -633.010,Z 581.325,A 0.000,B 0.000,C 90.000,E1 94.473} C_DIS
LIN {X -0.098,Y -635.262,Z 581.319,A 0.000,B 0.000,C 90.000,E1 93.498} C_DIS
LIN {X -0.072,Y -637.596,Z 581.312,A 0.000,B 0.000,C 90.000,E1 92.236} C_DIS
LIN {X 0.087,Y -638.427,Z 581.310,A 0.000,B 0.000,C 90.000,E1 91.718} C_DIS
LIN {X -0.257,Y -639.693,Z 581.304,A 0.000,B 0.000,C 90.000,E1 90.745} C_DIS
LIN {X 0.298,Y -640.396,Z 581.300,A 0.000,B 0.000,C 90.000,E1 89.943} C_DIS
LIN {X 0.222,Y -640.867,Z 581.296,A 0.000,B 0.000,C 90.000,E1 89.198} C_DIS
LIN {X 0.146,Y -641.096,Z 581.292,A 0.000,B 0.000,C 90.000,E1 88.453} C_DIS
LIN {X -0.146,Y -640.914,Z 581.286,A 0.000,B 0.000,C 90.000,E1 87.478} C_DIS
LIN {X -0.194,Y -640.593,Z 581.282,A 0.000,B 0.000,C 90.000,E1 86.731} C_DIS
LIN {X 0.152,Y -639.830,Z 581.276,A 0.000,B 0.000,C 90.000,E1 85.698} C_DIS
LIN {X -0.156,Y -638.739,Z 581.271,A 0.000,B 0.000,C 90.000,E1 84.723} C_DIS
LIN {X 0.212,Y -637.411,Z 581.265,A 0.000,B 0.000,C 90.000,E1 83.685} C_DIS
LIN {X 0.199,Y -636.239,Z 581.261,A 0.000,B 0.000,C 90.000,E1 82.932} C_DIS
LIN {X 0.095,Y -634.722,Z 581.257,A 0.000,B 0.000,C 90.000,E1 82.186} C_DIS
LIN {X 0.057,Y -633.134,Z 581.253,A 0.000,B 0.000,C 90.000,E1 81.432} C_DIS
LIN {X -0.189,Y -630.738,Z 581.247,A 0.000,B 0.000,C 90.000,E1 80.443} C_DIS
LIN {X -0.045,Y -627.437,Z 581.240,A 0.000,B 0.000,C 90.000,E1 79.162} C_DIS
LIN {X 0.035,Y -623.775,Z 581.233,A 0.000,B 0.000,C 90.000,E1 77.881} C_DIS
LIN {X 0.007,Y -621.369,Z 581.228,A 0.000,B 0.000,C 90.000,E1 77.117} C_DIS
LIN {X -0.268,Y -617.916,Z 581.223,A 0.000,B 0.000,C 90.000,E1 76.117} C_DIS
LIN {X -0.200,Y -615.122,Z 581.219,A 0.000,B 0.000,C 90.000,E1 75.338} C_DIS
LIN {X -0.315,Y -612.118,Z 581.214,A 0.000,B 0.000,C 90.000,E1 74.574} C_DIS
LIN {X -0.049,Y -609.931,Z 581.211,A 0.000,B 0.000,C 90.000,E1 74.031} C_DIS
LIN {X -0.269,Y -605.793,Z 581.206,A 0.000,B 0.000,C 90.000,E1 73.142} C_DIS
LIN {X -0.271,Y -602.670,Z 581.203,A 0.000,B 0.000,C 90.000,E1 72.489} C_DIS
LIN {X -0.172,Y -598.591,Z 581.198,A 0.000,B 0.000,C 90.000,E1 71.692} C_DIS
LIN {X -0.300,Y -594.208,Z 581.194,A 0.000,B 0.000,C 90.000,E1 70.913} C_DIS
LIN {X -0.104,Y -591.713,Z 581.192,A 0.000,B 0.000,C 90.000,E1 70.496} C_DIS
LIN {X 0.275,Y -589.354,Z 581.189,A 0.000,B 0.000,C 90.000,E1 70.061} C_DIS
